LIN {X 0,Y 467.201,Z 533.915,A -85,B 0,C 180,E1 -7658.87,E2 -7658.87} C_VEL
LIN {X 0,Y 467.55,Z 525.583,A -85,B 0,C 180,E1 -7660.173,E2 -7660.173} C_VEL
LIN {X 0,Y 467.994,Z 517.028,A -85,B 0,C 180,E1 -7661.258,E2 -7661.258} C_VEL
LIN {X 0,Y 468.515,Z 506.992,A -85,B 0,C 180,E1 -7662.295,E2 -7662.295} C_VEL
LIN {X 0,Y 468.892,Z 496.03,A -85,B 0,C 180,E1 -7663.213,E2 -7663.213} C_VEL
LIN {X 0,Y 469.41,Z 484.584,A -85,B 0,C 180,E1 -7663.971,E2 -7663.971} C_VEL
LIN {X 0,Y 469.934,Z 471.495,A -85,B 0,C 180,E1 -7664.618,E2 -7664.618} C_VEL
LIN {X 0,Y 468.494,Z 459.642,A -85,B 0,C 180,E1 -7665.094,E2 -7665.094} C_VEL
LIN {X 0,Y 466.973,Z 449.848,A -85,B 0,C 180,E1 -7665.416,E2 -7665.416} C_VEL
LIN {X 0,Y 467.157,Z 441.535,A -85,B 0,C 180,E1 -7668.596,E2 -7668.596} C_VEL
LIN {X 0,Y 467.367,Z 433.791,A -85,B 0,C 180,E1 -7671.618,E2 -7671.618} C_VEL
LIN {X 0,Y 467.629,Z 425.59,A -85,B 0,C 180,E1 -7674.886,E2 -7674.886} C_VEL
LIN {X 0,Y 467.958,Z 417.432,A -85,B 0,C 180,E1 -7678.235,E2 -7678.235} C_VEL
LIN {X 0,Y 468.288,Z 410.455,A -85,B 0,C 180,E1 -7681.19,E2 -7681.19} C_VEL
LIN {X 0,Y 468.615,Z 404.693,A -85,B 0,C 180,E1 -7683.704,E2 -7683.704} C_VEL
LIN {X 0,Y 468.72,Z 399.752,A -85,B 0,C 180,E1 -7685.935,E2 -7685.935} C_VEL
LIN {X 0,Y 468.166,Z 395.47,A -85,B 0,C 180,E1 -7687.987,E2 -7687.987} C_VEL
LIN {X 0,Y 467.621,Z 392.239,A -85,B 0,C 180,E1 -7689.628,E2 -7689.628} C_VEL
LIN {X 0,Y 467.588,Z 392.243,A -85,B 0,C 180,E1 -7692.567,E2 -7692.567} C_VEL
LIN {X 0,Y 467.567,Z 392.245,A -85,B 0,C 180,E1 -7695.052,E2 -7695.052} C_VEL
LIN {X 0,Y 467.59,Z 392.242,A -85,B 0,C 180,E1 -7697.44,E2 -7697.44} C_VEL
LIN {X 0,Y 467.577,Z 392.245,A -85,B 0,C 180,E1 -7700.855,E2 -7700.855} C_VEL
LIN {X 0,Y 467.562,Z 392.244,A -85,B 0,C 180,E1 -7704.261,E2 -7704.261} C_VEL
LIN {X 0,Y 467.58,Z 392.243,A -85,B 0,C 180,E1 -7707.321,E2 -7707.321} C_VEL
LIN {X 0,Y 467.571,Z 392.244,A -85,B 0,C 180,E1 -7710.667,E2 -7710.667} C_VEL
LIN {X 0,Y 467.617,Z 392.238,A -85,B 0,C 180,E1 -7713.2,E2 -7713.2} C_VEL
LIN {X 0,Y 467.593,Z 392.241,A -85,B 0,C 180,E1 -7716.468,E2 -7716.468} C_VEL
LIN {X 0,Y 467.623,Z 392.237,A -85,B 0,C 180,E1 -7719.777,E2 -7719.777} C_VEL
LIN {X 0,Y 467.607,Z 392.24,A -85,B 0,C 180,E1 -7722.507,E2 -7722.507} C_VEL
LIN {X 0,Y 467.607,Z 392.24,A -85,B 0,C 180,E1 -7725.196,E2 -7725.196} C_VEL
LIN {X 0,Y 467.656,Z 392.233,A -85,B 0,C 180,E1 -7727.854,E2 -7727.854} C_VEL
LIN {X 0,Y 467.682,Z 392.231,A -85,B 0,C 180,E1 -7731.357,E2 -7731.357} C_VEL
LIN {X 0,Y 467.744,Z 392.221,A -85,B 0,C 180,E1 -7733.963,E2 -7733.963} C_VEL
LIN {X 0,Y 467.859,Z 392.209,A -85,B 0,C 180,E1 -7737.417,E2 -7737.417} C_VEL
LIN {X 0,Y 467.882,Z 392.204,A -85,B 0,C 180,E1 -7740,E2 -7740} C_VEL
LIN {X 0,Y 467.859,Z 392.21,A -85,B 0,C 180,E1 -7742.583,E2 -7742.583} C_VEL
LIN {X 0,Y 467.743,Z 392.222,A -85,B 0,C 180,E1 -7746.037,E2 -7746.037} C_VEL
LIN {X 0,Y 467.682,Z 392.231,A -85,B 0,C 180,E1 -7748.643,E2 -7748.643} C_VEL
LIN {X 0,Y 467.656,Z 392.233,A -85,B 0,C 180,E1 -7752.145,E2 -7752.145} C_VEL
LIN {X 0,Y 467.639,Z 392.234,A -85,B 0,C 180,E1 -7755.695,E2 -7755.695} C_VEL
LIN {X 0,Y 467.618,Z 392.239,A -85,B 0,C 180,E1 -7758.764,E2 -7758.764} C_VEL
LIN {X 0,Y 467.581,Z 392.244,A -85,B 0,C 180,E1 -7761.268,E2 -7761.268} C_VEL
LIN {X 0,Y 467.572,Z 392.243,A -85,B 0,C 180,E1 -7763.943,E2 -7763.943} C_VEL
LIN {X 0,Y 467.617,Z 392.238,A -85,B 0,C 180,E1 -7766.8,E2 -7766.8} C_VEL
LIN {X 0,Y 467.554,Z 392.245,A -85,B 0,C 180,E1 -7769.738,E2 -7769.738} C_VEL
LIN {X 0,Y 467.584,Z 392.243,A -85,B 0,C 180,E1 -7772.758,E2 -7772.758} C_VEL
LIN {X 0,Y 467.557,Z 392.245,A -85,B 0,C 180,E1 -7775.889,E2 -7775.889} C_VEL
LIN {X 0,Y 467.576,Z 392.244,A -85,B 0,C 180,E1 -7779.145,E2 -7779.145} C_VEL
LIN {X 0,Y 467.587,Z 392.242,A -85,B 0,C 180,E1 -7782.567,E2 -7782.567} C_VEL
LIN {X 0,Y 467.567,Z 392.245,A -85,B 0,C 180,E1 -7785.053,E2 -7785.053} C_VEL
LIN {X 0,Y 467.59,Z 392.241,A -85,B 0,C 180,E1 -7787.44,E2 -7787.44} C_VEL
LIN {X 0,Y 467.583,Z 392.243,A -85,B 0,C 180,E1 -7790.855,E2 -7790.855} C_VEL
LIN {X 0,Y 467.564,Z 392.245,A -85,B 0,C 180,E1 -7794.26,E2 -7794.26} C_VEL
LIN {X 0,Y 467.583,Z 392.242,A -85,B 0,C 180,E1 -7797.321,E2 -7797.321} C_VEL
LIN {X 0,Y 467.572,Z 392.245,A -85,B 0,C 180,E1 -7800.667,E2 -7800.667} C_VEL
LIN {X 0,Y 467.618,Z 392.238,A -85,B 0,C 180,E1 -7803.2,E2 -7803.2} C_VEL
LIN {X 0,Y 467.595,Z 392.241,A -85,B 0,C 180,E1 -7806.468,E2 -7806.468} C_VEL
LIN {X 0,Y 467.625,Z 392.236,A -85,B 0,C 180,E1 -7809.777,E2 -7809.777} C_VEL
LIN {X 0,Y 467.609,Z 392.24,A -85,B 0,C 180,E1 -7812.507,E2 -7812.507} C_VEL
LIN {X 0,Y 467.599,Z 392.239,A -85,B 0,C 180,E1 -7815.416,E2 -7815.416} C_VEL
LIN {X 0,Y 466.929,Z 392.325,A -85,B 0,C 180,E1 -7816.135,E2 -7816.135} C_VEL
LIN {X 0,Y 464.085,Z 392.677,A -85,B 0,C 180,E1 -7817.303,E2 -7817.303} C_VEL
LIN {X 0,Y 461.686,Z 392.977,A -85,B 0,C 180,E1 -7818.245,E2 -7818.245} C_VEL
LIN {X 0,Y 460.659,Z 393.104,A -85,B 0,C 180,E1 -7818.973,E2 -7818.973} C_VEL
LIN {X 0,Y 460.576,Z 393.112,A -85,B 0,C 180,E1 -7819.219,E2 -7819.219} C_VEL
LIN {X 0,Y 460.723,Z 393.098,A -85,B 0,C 180,E1 -7822.538,E2 -7822.538} C_VEL
LIN {X 0,Y 460.699,Z 393.1,A -85,B 0,C 180,E1 -7824.748,E2 -7824.748} C_VEL
LIN {X 0,Y 460.802,Z 393.086,A -85,B 0,C 180,E1 -7827.377,E2 -7827.377} C_VEL
LIN {X 0,Y 460.855,Z 393.081,A -85,B 0,C 180,E1 -7830,E2 -7830} C_VEL
LIN {X 0,Y 460.826,Z 393.084,A -85,B 0,C 180,E1 -7832.622,E2 -7832.622} C_VEL
LIN {X 0,Y 460.679,Z 393.103,A -85,B 0,C 180,E1 -7836.13,E2 -7836.13} C_VEL
LIN {X 0,Y 460.387,Z 393.141,A -85,B 0,C 180,E1 -7838.78,E2 -7838.78} C_VEL
LIN {X 0,Y 460.288,Z 393.863,A -85,B 0,C 180,E1 -7839.669,E2 -7839.669} C_VEL
LIN {X 0,Y 460.2,Z 397.277,A -85,B 0,C 180,E1 -7842.345,E2 -7842.345} C_VEL
LIN {X 0,Y 460.068,Z 401.733,A -85,B 0,C 180,E1 -7845.764,E2 -7845.764} C_VEL
LIN {X 0,Y 459.93,Z 405.642,A -85,B 0,C 180,E1 -7848.716,E2 -7848.716} C_VEL
LIN {X 0,Y 459.788,Z 409.438,A -85,B 0,C 180,E1 -7851.521,E2 -7851.521} C_VEL
LIN {X 0,Y 459.726,Z 413.312,A -85,B 0,C 180,E1 -7854.378,E2 -7854.378} C_VEL
LIN {X 0,Y 459.679,Z 417.601,A -85,B 0,C 180,E1 -7857.454,E2 -7857.454} C_VEL
LIN {X 0,Y 462.867,Z 432.273,A -85,B 0,C 180,E1 -7858.027,E2 -7858.027} C_VEL
LIN {X 0,Y 463.264,Z 437.27,A -85,B 0,C 180,E1 -7858.249,E2 -7858.249} C_VEL
LIN {X 0,Y 462.774,Z 449.809,A -85,B 0,C 180,E1 -7858.889,E2 -7858.889} C_VEL
LIN {X 0,Y 462.259,Z 460.524,A -85,B 0,C 180,E1 -7859.607,E2 -7859.607} C_VEL
LIN {X 0,Y 461.801,Z 471.37,A -85,B 0,C 180,E1 -7860.525,E2 -7860.525} C_VEL
LIN {X 0,Y 461.318,Z 481.28,A -85,B 0,C 180,E1 -7861.56,E2 -7861.56} C_VEL
LIN {X 0,Y 460.844,Z 490.462,A -85,B 0,C 180,E1 -7862.743,E2 -7862.743} C_VEL
LIN {X 0,Y 460.4,Z 499.041,A -85,B 0,C 180,E1 -7864.123,E2 -7864.123} C_VEL
LIN {X 0,Y 460.06,Z 505.812,A -85,B 0,C 180,E1 -7865.485,E2 -7865.485} C_VEL
LIN {X 0,Y 459.849,Z 511.567,A -85,B 0,C 180,E1 -7866.968,E2 -7866.968} C_VEL
LIN {X 0,Y 459.685,Z 515.328,A -85,B 0,C 180,E1 -7868.225,E2 -7868.225} C_VEL
LIN {X 0,Y 459.574,Z 517.956,A -85,B 0,C 180,E1 -7869.392,E2 -7869.392} C_VEL
LIN {X 0,Y 459.493,Z 519.215,A -85,B 0,C 180,E1 -7870.115,E2 -7870.115} C_VEL
LIN {X 0,Y 459.433,Z 520.788,A -85,B 0,C 180,E1 -7871.448,E2 -7871.448} C_VEL
LIN {X 0,Y 459.462,Z 521.432,A -85,B 0,C 180,E1 -7872.759,E2 -7872.759} C_VEL
LIN {X 0,Y 459.474,Z 521.217,A -85,B 0,C 180,E1 -7874.036,E2 -7874.036} C_VEL
LIN {X 0,Y 459.498,Z 520.204,A -85,B 0,C 180,E1 -7875.286,E2 -7875.286} C_VEL
LIN {X 0,Y 459.593,Z 518.401,A -85,B 0,C 180,E1 -7876.518,E2 -7876.518} C_VEL
LIN {X 0,Y 459.735,Z 514.685,A -85,B 0,C 180,E1 -7878.149,E2 -7878.149} C_VEL
LIN {X 0,Y 459.919,Z 509.247,A -85,B 0,C 180,E1 -7879.821,E2 -7879.821} C_VEL
LIN {X 0,Y 460.22,Z 503.109,A -85,B 0,C 180,E1 -7881.236,E2 -7881.236} C_VEL
LIN {X 0,Y 460.581,Z 496.18,A -85,B 0,C 180,E1 -7882.51,E2 -7882.51} C_VEL
LIN {X 0,Y 461.062,Z 486.859,A -85,B 0,C 180,E1 -7883.888,E2 -7883.888} C_VEL
LIN {X 0,Y 461.597,Z 477.131,A -85,B 0,C 180,E1 -7885.034,E2 -7885.034} C_VEL
LIN {X 0,Y 462.139,Z 466.904,A -85,B 0,C 180,E1 -7886.007,E2 -7886.007} C_VEL
LIN {X 0,Y 462.597,Z 456.021,A -85,B 0,C 180,E1 -7886.843,E2 -7886.843} C_VEL
LIN {X 0,Y 463.118,Z 444.532,A -85,B 0,C 180,E1 -7887.532,E2 -7887.532} C_VEL
LIN {X 0,Y 463.321,Z 434.551,A -85,B 0,C 180,E1 -7887.997,E2 -7887.997} C_VEL
LIN {X 0,Y 460.593,Z 421.943,A -85,B 0,C 180,E1 -7888.525,E2 -7888.525} C_VEL
LIN {X 0,Y 459.753,Z 418.131,A -85,B 0,C 180,E1 -7888.669,E2 -7888.669} C_VEL
LIN {X 0,Y 459.786,Z 414.027,A -85,B 0,C 180,E1 -7891.716,E2 -7891.716} C_VEL
LIN {X 0,Y 459.956,Z 410.111,A -85,B 0,C 180,E1 -7894.67,E2 -7894.67} C_VEL
LIN {X 0,Y 460.056,Z 406.354,A -85,B 0,C 180,E1 -7897.548,E2 -7897.548} C_VEL
LIN {X 0,Y 460.159,Z 402.747,A -85,B 0,C 180,E1 -7900.366,E2 -7900.366} C_VEL
LIN {X 0,Y 460.271,Z 399.284,A -85,B 0,C 180,E1 -7903.135,E2 -7903.135} C_VEL
LIN {X 0,Y 460.374,Z 395.891,A -85,B 0,C 180,E1 -7905.862,E2 -7905.862} C_VEL
LIN {X 0,Y 460.468,Z 393.714,A -85,B 0,C 180,E1 -7907.662,E2 -7907.662} C_VEL
LIN {X 0,Y 460.519,Z 393.124,A -85,B 0,C 180,E1 -7908.557,E2 -7908.557} C_VEL
LIN {X 0,Y 460.624,Z 393.114,A -85,B 0,C 180,E1 -7911.224,E2 -7911.224} C_VEL
LIN {X 0,Y 460.706,Z 393.099,A -85,B 0,C 180,E1 -7913.87,E2 -7913.87} C_VEL
LIN {X 0,Y 460.821,Z 393.086,A -85,B 0,C 180,E1 -7917.378,E2 -7917.378} C_VEL
LIN {X 0,Y 460.849,Z 393.082,A -85,B 0,C 180,E1 -7920,E2 -7920} C_VEL
LIN {X 0,Y 460.82,Z 393.084,A -85,B 0,C 180,E1 -7922.622,E2 -7922.622} C_VEL
LIN {X 0,Y 460.706,Z 393.1,A -85,B 0,C 180,E1 -7926.13,E2 -7926.13} C_VEL
LIN {X 0,Y 460.625,Z 393.11,A -85,B 0,C 180,E1 -7928.776,E2 -7928.776} C_VEL
LIN {X 0,Y 460.609,Z 393.112,A -85,B 0,C 180,E1 -7932.445,E2 -7932.445} C_VEL
LIN {X 0,Y 460.596,Z 393.113,A -85,B 0,C 180,E1 -7935.998,E2 -7935.998} C_VEL
LIN {X 0,Y 460.567,Z 393.116,A -85,B 0,C 180,E1 -7938.902,E2 -7938.902} C_VEL
LIN {X 0,Y 460.512,Z 393.124,A -85,B 0,C 180,E1 -7941.486,E2 -7941.486} C_VEL
LIN {X 0,Y 460.539,Z 393.118,A -85,B 0,C 180,E1 -7944.333,E2 -7944.333} C_VEL
LIN {X 0,Y 460.581,Z 393.115,A -85,B 0,C 180,E1 -7947.243,E2 -7947.243} C_VEL
LIN {X 0,Y 460.524,Z 393.122,A -85,B 0,C 180,E1 -7950.239,E2 -7950.239} C_VEL
LIN {X 0,Y 460.526,Z 393.122,A -85,B 0,C 180,E1 -7953.325,E2 -7953.325} C_VEL
LIN {X 0,Y 460.477,Z 393.129,A -85,B 0,C 180,E1 -7956.53,E2 -7956.53} C_VEL
LIN {X 0,Y 460.576,Z 393.117,A -85,B 0,C 180,E1 -7959.858,E2 -7959.858} C_VEL
LIN {X 0,Y 460.511,Z 393.125,A -85,B 0,C 180,E1 -7962.901,E2 -7962.901} C_VEL
LIN {X 0,Y 460.509,Z 393.124,A -85,B 0,C 180,E1 -7965.831,E2 -7965.831} C_VEL
LIN {X 0,Y 460.541,Z 393.119,A -85,B 0,C 180,E1 -7968.991,E2 -7968.991} C_VEL
LIN {X 0,Y 460.58,Z 393.173,A -85,B 0,C 180,E1 -7969.799,E2 -7969.799} C_VEL
LIN {X 0,Y 461.533,Z 399.106,A -85,B 0,C 180,E1 -7973.024,E2 -7973.024} C_VEL
LIN {X 0,Y 461.753,Z 403.631,A -85,B 0,C 180,E1 -7975.275,E2 -7975.275} C_VEL
LIN {X 0,Y 461.39,Z 408.979,A -85,B 0,C 180,E1 -7977.784,E2 -7977.784} C_VEL
LIN {X 0,Y 460.976,Z 415.748,A -85,B 0,C 180,E1 -7980.8,E2 -7980.8} C_VEL
LIN {X 0,Y 460.62,Z 423.684,A -85,B 0,C 180,E1 -7984.185,E2 -7984.185} C_VEL
LIN {X 0,Y 460.34,Z 431.917,A -85,B 0,C 180,E1 -7987.563,E2 -7987.563} C_VEL
LIN {X 0,Y 460.079,Z 440.121,A -85,B 0,C 180,E1 -7990.827,E2 -7990.827} C_VEL
LIN {X 0,Y 459.905,Z 448.373,A -85,B 0,C 180,E1 -7994.035,E2 -7994.035} C_VEL
LIN {X 0,Y 459.859,Z 449.138,A -85,B 0,C 180,E1 -7994.329,E2 -7994.329} C_VEL
LIN {X 0,Y 462.172,Z 464.362,A -85,B 0,C 180,E1 -7994.857,E2 -7994.857} C_VEL
LIN {X 0,Y 463.01,Z 472.453,A -85,B 0,C 180,E1 -7995.215,E2 -7995.215} C_VEL
LIN {X 0,Y 462.524,Z 484.144,A -85,B 0,C 180,E1 -7995.818,E2 -7995.818} C_VEL
LIN {X 0,Y 461.969,Z 495.547,A -85,B 0,C 180,E1 -7996.586,E2 -7996.586} C_VEL
LIN {X 0,Y 461.437,Z 506.673,A -85,B 0,C 180,E1 -7997.531,E2 -7997.531} C_VEL
LIN {X 0,Y 460.977,Z 516.553,A -85,B 0,C 180,E1 -7998.569,E2 -7998.569} C_VEL
LIN {X 0,Y 460.496,Z 525.123,A -85,B 0,C 180,E1 -7999.67,E2 -7999.67} C_VEL
LIN {X 0,Y 460.129,Z 533.481,A -85,B 0,C 180,E1 -8000.993,E2 -8000.993} C_VEL
LIN {X 0,Y 459.883,Z 540.226,A -85,B 0,C 180,E1 -8002.316,E2 -8002.316} C_VEL
LIN {X 0,Y 459.674,Z 546.407,A -85,B 0,C 180,E1 -8003.857,E2 -8003.857} C_VEL
LIN {X 0,Y 459.621,Z 550.425,A -85,B 0,C 180,E1 -8005.176,E2 -8005.176} C_VEL
LIN {X 0,Y 459.588,Z 553.396,A -85,B 0,C 180,E1 -8006.494,E2 -8006.494} C_VEL
LIN {X 0,Y 459.585,Z 554.812,A -85,B 0,C 180,E1 -8007.371,E2 -8007.371} C_VEL
LIN {X 0,Y 459.552,Z 556.446,A -85,B 0,C 180,E1 -8009.124,E2 -8009.124} C_VEL
LIN {X 0,Y 459.53,Z 556.67,A -85,B 0,C 180,E1 -8010,E2 -8010} C_VEL
LIN {X 0,Y 459.552,Z 556.459,A -85,B 0,C 180,E1 -8010.877,E2 -8010.877} C_VEL
LIN {X 0,Y 459.585,Z 554.857,A -85,B 0,C 180,E1 -8012.63,E2 -8012.63} C_VEL
LIN {X 0,Y 459.588,Z 553.453,A -85,B 0,C 180,E1 -8013.507,E2 -8013.507} C_VEL
LIN {X 0,Y 459.621,Z 550.502,A -85,B 0,C 180,E1 -8014.825,E2 -8014.825} C_VEL
LIN {X 0,Y 459.715,Z 545.46,A -85,B 0,C 180,E1 -8016.431,E2 -8016.431} C_VEL
LIN {X 0,Y 459.909,Z 539.328,A -85,B 0,C 180,E1 -8017.905,E2 -8017.905} C_VEL
LIN {X 0,Y 460.226,Z 532.379,A -85,B 0,C 180,E1 -8019.227,E2 -8019.227} C_VEL
LIN {X 0,Y 460.581,Z 523.669,A -85,B 0,C 180,E1 -8020.551,E2 -8020.551} C_VEL
LIN {X 0,Y 461.103,Z 514.757,A -85,B 0,C 180,E1 -8021.651,E2 -8021.651} C_VEL
LIN {X 0,Y 461.615,Z 504.111,A -85,B 0,C 180,E1 -8022.724,E2 -8022.724} C_VEL
LIN {X 0,Y 462.104,Z 492.682,A -85,B 0,C 180,E1 -8023.635,E2 -8023.635} C_VEL
LIN {X 0,Y 462.691,Z 480.292,A -85,B 0,C 180,E1 -8024.402,E2 -8024.402} C_VEL
LIN {X 0,Y 463.053,Z 471.128,A -85,B 0,C 180,E1 -8024.84,E2 -8024.84} C_VEL
LIN {X 0,Y 461.181,Z 457.798,A -85,B 0,C 180,E1 -8025.384,E2 -8025.384} C_VEL
LIN {X 0,Y 459.908,Z 449.618,A -85,B 0,C 180,E1 -8025.642,E2 -8025.642} C_VEL
LIN {X 0,Y 460.117,Z 440.704,A -85,B 0,C 180,E1 -8029.126,E2 -8029.126} C_VEL
LIN {X 0,Y 460.325,Z 433.575,A -85,B 0,C 180,E1 -8031.966,E2 -8031.966} C_VEL
LIN {X 0,Y 460.609,Z 425.402,A -85,B 0,C 180,E1 -8035.292,E2 -8035.292} C_VEL
LIN {X 0,Y 460.971,Z 417.26,A -85,B 0,C 180,E1 -8038.702,E2 -8038.702} C_VEL
LIN {X 0,Y 461.291,Z 410.929,A -85,B 0,C 180,E1 -8041.439,E2 -8041.439} C_VEL
LIN {X 0,Y 461.737,Z 403.563,A -85,B 0,C 180,E1 -8044.722,E2 -8044.722} C_VEL
LIN {X 0,Y 461.531,Z 398.786,A -85,B 0,C 180,E1 -8046.977,E2 -8046.977} C_VEL
LIN {X 0,Y 460.574,Z 393.117,A -85,B 0,C 180,E1 -8049.858,E2 -8049.858} C_VEL
LIN {X 0,Y 460.514,Z 393.123,A -85,B 0,C 180,E1 -8052.9,E2 -8052.9} C_VEL
LIN {X 0,Y 460.51,Z 393.125,A -85,B 0,C 180,E1 -8055.831,E2 -8055.831} C_VEL
LIN {X 0,Y 460.532,Z 393.121,A -85,B 0,C 180,E1 -8058.989,E2 -8058.989} C_VEL
LIN {X 0,Y 460.525,Z 393.122,A -85,B 0,C 180,E1 -8061.267,E2 -8061.267} C_VEL
LIN {X 0,Y 460.512,Z 393.123,A -85,B 0,C 180,E1 -8064.554,E2 -8064.554} C_VEL
LIN {X 0,Y 460.531,Z 393.121,A -85,B 0,C 180,E1 -8067.715,E2 -8067.715} C_VEL
LIN {X 0,Y 460.541,Z 393.12,A -85,B 0,C 180,E1 -8070.769,E2 -8070.769} C_VEL
LIN {X 0,Y 460.564,Z 393.116,A -85,B 0,C 180,E1 -8073.735,E2 -8073.735} C_VEL
LIN {X 0,Y 460.547,Z 393.119,A -85,B 0,C 180,E1 -8076.624,E2 -8076.624} C_VEL
LIN {X 0,Y 460.552,Z 393.119,A -85,B 0,C 180,E1 -8079.453,E2 -8079.453} C_VEL
LIN {X 0,Y 460.558,Z 393.117,A -85,B 0,C 180,E1 -8082.23,E2 -8082.23} C_VEL
LIN {X 0,Y 460.566,Z 393.117,A -85,B 0,C 180,E1 -8084.965,E2 -8084.965} C_VEL
LIN {X 0,Y 460.611,Z 393.111,A -85,B 0,C 180,E1 -8088.559,E2 -8088.559} C_VEL
LIN {X 0,Y 460.696,Z 393.099,A -85,B 0,C 180,E1 -8092.108,E2 -8092.108} C_VEL
LIN {X 0,Y 460.696,Z 393.1,A -85,B 0,C 180,E1 -8094.748,E2 -8094.748} C_VEL
LIN {X 0,Y 460.8,Z 393.088,A -85,B 0,C 180,E1 -8097.377,E2 -8097.377} C_VEL
LIN {X 0,Y 460.853,Z 393.08,A -85,B 0,C 180,E1 -8100,E2 -8100} C_VEL
LIN {X 0,Y 460.8,Z 393.089,A -85,B 0,C 180,E1 -8102.622,E2 -8102.622} C_VEL
LIN {X 0,Y 460.71,Z 393.098,A -85,B 0,C 180,E1 -8106.13,E2 -8106.13} C_VEL
LIN {X 0,Y 460.629,Z 393.109,A -85,B 0,C 180,E1 -8108.776,E2 -8108.776} C_VEL
LIN {X 0,Y 460.614,Z 393.111,A -85,B 0,C 180,E1 -8112.445,E2 -8112.445} C_VEL
LIN {X 0,Y 460.601,Z 393.111,A -85,B 0,C 180,E1 -8115.998,E2 -8115.998} C_VEL
LIN {X 0,Y 460.571,Z 393.117,A -85,B 0,C 180,E1 -8118.902,E2 -8118.902} C_VEL
LIN {X 0,Y 460.516,Z 393.122,A -85,B 0,C 180,E1 -8121.486,E2 -8121.486} C_VEL
LIN {X 0,Y 460.542,Z 393.12,A -85,B 0,C 180,E1 -8124.332,E2 -8124.332} C_VEL
LIN {X 0,Y 460.573,Z 393.116,A -85,B 0,C 180,E1 -8127.244,E2 -8127.244} C_VEL
LIN {X 0,Y 460.511,Z 393.124,A -85,B 0,C 180,E1 -8130.24,E2 -8130.24} C_VEL
LIN {X 0,Y 460.53,Z 393.121,A -85,B 0,C 180,E1 -8133.325,E2 -8133.325} C_VEL
LIN {X 0,Y 460.479,Z 393.127,A -85,B 0,C 180,E1 -8136.529,E2 -8136.529} C_VEL
LIN {X 0,Y 460.528,Z 393.12,A -85,B 0,C 180,E1 -8139.863,E2 -8139.863} C_VEL
LIN {X 0,Y 460.514,Z 393.124,A -85,B 0,C 180,E1 -8142.9,E2 -8142.9} C_VEL
LIN {X 0,Y 460.51,Z 393.123,A -85,B 0,C 180,E1 -8145.831,E2 -8145.831} C_VEL
LIN {X 0,Y 460.532,Z 393.121,A -85,B 0,C 180,E1 -8148.989,E2 -8148.989} C_VEL
LIN {X 0,Y 460.527,Z 393.121,A -85,B 0,C 180,E1 -8151.267,E2 -8151.267} C_VEL
LIN {X 0,Y 460.514,Z 393.124,A -85,B 0,C 180,E1 -8154.555,E2 -8154.555} C_VEL
LIN {X 0,Y 460.533,Z 393.12,A -85,B 0,C 180,E1 -8157.716,E2 -8157.716} C_VEL
LIN {X 0,Y 460.542,Z 393.121,A -85,B 0,C 180,E1 -8160.769,E2 -8160.769} C_VEL
LIN {X 0,Y 460.565,Z 393.116,A -85,B 0,C 180,E1 -8163.735,E2 -8163.735} C_VEL
LIN {X 0,Y 460.548,Z 393.12,A -85,B 0,C 180,E1 -8166.624,E2 -8166.624} C_VEL
LIN {X 0,Y 460.553,Z 393.117,A -85,B 0,C 180,E1 -8169.453,E2 -8169.453} C_VEL
LIN {X 0,Y 460.559,Z 393.117,A -85,B 0,C 180,E1 -8172.23,E2 -8172.23} C_VEL
LIN {X 0,Y 460.568,Z 393.117,A -85,B 0,C 180,E1 -8174.965,E2 -8174.965} C_VEL
LIN {X 0,Y 460.612,Z 393.112,A -85,B 0,C 180,E1 -8178.559,E2 -8178.559} C_VEL
LIN {X 0,Y 460.576,Z 393.112,A -85,B 0,C 180,E1 -8179.219,E2 -8179.219} C_VEL
LIN {X 0,Y 459.92,Z 393.197,A -85,B 0,C 180,E1 -8179.949,E2 -8179.949} C_VEL
LIN {X 0,Y 457.105,Z 393.547,A -85,B 0,C 180,E1 -8181.136,E2 -8181.136} C_VEL
LIN {X 0,Y 454.728,Z 393.844,A -85,B 0,C 180,E1 -8182.093,E2 -8182.093} C_VEL
LIN {X 0,Y 453.717,Z 393.969,A -85,B 0,C 180,E1 -8182.832,E2 -8182.832} C_VEL
LIN {X 0,Y 453.64,Z 393.977,A -85,B 0,C 180,E1 -8183.082,E2 -8183.082} C_VEL
LIN {X 0,Y 453.673,Z 393.976,A -85,B 0,C 180,E1 -8184.666,E2 -8184.666} C_VEL
LIN {X 0,Y 453.746,Z 393.965,A -85,B 0,C 180,E1 -8187.336,E2 -8187.336} C_VEL
LIN {X 0,Y 453.825,Z 393.956,A -85,B 0,C 180,E1 -8190,E2 -8190} C_VEL
LIN {X 0,Y 453.767,Z 393.964,A -85,B 0,C 180,E1 -8192.663,E2 -8192.663} C_VEL
LIN {X 0,Y 453.641,Z 393.979,A -85,B 0,C 180,E1 -8196.225,E2 -8196.225} C_VEL
LIN {X 0,Y 453.313,Z 394.022,A -85,B 0,C 180,E1 -8198.919,E2 -8198.919} C_VEL
LIN {X 0,Y 453.168,Z 396.002,A -85,B 0,C 180,E1 -8200.725,E2 -8200.725} C_VEL
LIN {X 0,Y 453.098,Z 399.471,A -85,B 0,C 180,E1 -8203.454,E2 -8203.454} C_VEL
LIN {X 0,Y 452.935,Z 403.058,A -85,B 0,C 180,E1 -8206.218,E2 -8206.218} C_VEL
LIN {X 0,Y 452.821,Z 406.756,A -85,B 0,C 180,E1 -8209.021,E2 -8209.021} C_VEL
LIN {X 0,Y 452.7,Z 410.561,A -85,B 0,C 180,E1 -8211.875,E2 -8211.875} C_VEL
LIN {X 0,Y 452.651,Z 414.507,A -85,B 0,C 180,E1 -8214.784,E2 -8214.784} C_VEL
LIN {X 0,Y 452.599,Z 417.813,A -85,B 0,C 180,E1 -8217.2,E2 -8217.2} C_VEL
LIN {X 0,Y 456.011,Z 433.552,A -85,B 0,C 180,E1 -8217.843,E2 -8217.843} C_VEL
LIN {X 0,Y 456.383,Z 437.928,A -85,B 0,C 180,E1 -8218.047,E2 -8218.047} C_VEL
LIN {X 0,Y 455.875,Z 449.998,A -85,B 0,C 180,E1 -8218.674,E2 -8218.674} C_VEL
LIN {X 0,Y 455.31,Z 461.602,A -85,B 0,C 180,E1 -8219.472,E2 -8219.472} C_VEL
LIN {X 0,Y 454.862,Z 471.75,A -85,B 0,C 180,E1 -8220.35,E2 -8220.35} C_VEL
LIN {X 0,Y 454.317,Z 481.996,A -85,B 0,C 180,E1 -8221.441,E2 -8221.441} C_VEL
LIN {X 0,Y 453.868,Z 490.484,A -85,B 0,C 180,E1 -8222.553,E2 -8222.553} C_VEL
LIN {X 0,Y 453.411,Z 498.904,A -85,B 0,C 180,E1 -8223.918,E2 -8223.918} C_VEL
LIN {X 0,Y 453.054,Z 505.74,A -85,B 0,C 180,E1 -8225.298,E2 -8225.298} C_VEL
LIN {X 0,Y 452.824,Z 511.214,A -85,B 0,C 180,E1 -8226.694,E2 -8226.694} C_VEL
LIN {X 0,Y 452.595,Z 516.179,A -85,B 0,C 180,E1 -8228.398,E2 -8228.398} C_VEL
LIN {X 0,Y 452.466,Z 518.637,A -85,B 0,C 180,E1 -8229.556,E2 -8229.556} C_VEL
LIN {X 0,Y 452.356,Z 520.366,A -85,B 0,C 180,E1 -8230.732,E2 -8230.732} C_VEL
LIN {X 0,Y 452.341,Z 521.396,A -85,B 0,C 180,E1 -8231.919,E2 -8231.919} C_VEL
LIN {X 0,Y 452.387,Z 521.748,A -85,B 0,C 180,E1 -8233.121,E2 -8233.121} C_VEL
LIN {X 0,Y 452.379,Z 521.317,A -85,B 0,C 180,E1 -8234.386,E2 -8234.386} C_VEL
LIN {X 0,Y 452.436,Z 520.069,A -85,B 0,C 180,E1 -8235.652,E2 -8235.652} C_VEL
LIN {X 0,Y 452.535,Z 518.052,A -85,B 0,C 180,E1 -8236.895,E2 -8236.895} C_VEL
LIN {X 0,Y 452.66,Z 515.102,A -85,B 0,C 180,E1 -8238.179,E2 -8238.179} C_VEL
LIN {X 0,Y 452.815,Z 511.032,A -85,B 0,C 180,E1 -8239.508,E2 -8239.508} C_VEL
LIN {X 0,Y 453.099,Z 505.737,A -85,B 0,C 180,E1 -8240.854,E2 -8240.854} C_VEL
LIN {X 0,Y 453.438,Z 498.942,A -85,B 0,C 180,E1 -8242.228,E2 -8242.228} C_VEL
LIN {X 0,Y 453.859,Z 491.28,A -85,B 0,C 180,E1 -8243.48,E2 -8243.48} C_VEL
LIN {X 0,Y 454.365,Z 482.232,A -85,B 0,C 180,E1 -8244.681,E2 -8244.681} C_VEL
LIN {X 0,Y 454.967,Z 471.593,A -85,B 0,C 180,E1 -8245.813,E2 -8245.813} C_VEL
LIN {X 0,Y 455.482,Z 461.711,A -85,B 0,C 180,E1 -8246.664,E2 -8246.664} C_VEL
LIN {X 0,Y 455.966,Z 450.849,A -85,B 0,C 180,E1 -8247.417,E2 -8247.417} C_VEL
LIN {X 0,Y 456.432,Z 439.403,A -85,B 0,C 180,E1 -8248.03,E2 -8248.03} C_VEL
LIN {X 0,Y 456.379,Z 434.991,A -85,B 0,C 180,E1 -8248.23,E2 -8248.23} C_VEL
LIN {X 0,Y 453.535,Z 422.238,A -85,B 0,C 180,E1 -8248.779,E2 -8248.779} C_VEL
LIN {X 0,Y 452.679,Z 418.434,A -85,B 0,C 180,E1 -8248.918,E2 -8248.918} C_VEL
LIN {X 0,Y 452.766,Z 414.026,A -85,B 0,C 180,E1 -8252.246,E2 -8252.246} C_VEL
LIN {X 0,Y 452.897,Z 410.115,A -85,B 0,C 180,E1 -8255.23,E2 -8255.23} C_VEL
LIN {X 0,Y 453.049,Z 405.876,A -85,B 0,C 180,E1 -8258.551,E2 -8258.551} C_VEL
LIN {X 0,Y 453.174,Z 401.64,A -85,B 0,C 180,E1 -8261.931,E2 -8261.931} C_VEL
LIN {X 0,Y 453.304,Z 398.22,A -85,B 0,C 180,E1 -8264.718,E2 -8264.718} C_VEL
LIN {X 0,Y 453.443,Z 394.834,A -85,B 0,C 180,E1 -8267.537,E2 -8267.537} C_VEL
LIN {X 0,Y 453.462,Z 394.004,A -85,B 0,C 180,E1 -8268.376,E2 -8268.376} C_VEL
LIN {X 0,Y 453.586,Z 393.99,A -85,B 0,C 180,E1 -8271.087,E2 -8271.087} C_VEL
LIN {X 0,Y 453.673,Z 393.976,A -85,B 0,C 180,E1 -8273.775,E2 -8273.775} C_VEL
LIN {X 0,Y 453.762,Z 393.966,A -85,B 0,C 180,E1 -8277.337,E2 -8277.337} C_VEL
LIN {X 0,Y 453.82,Z 393.957,A -85,B 0,C 180,E1 -8280,E2 -8280} C_VEL
LIN {X 0,Y 453.761,Z 393.964,A -85,B 0,C 180,E1 -8282.663,E2 -8282.663} C_VEL
LIN {X 0,Y 453.674,Z 393.976,A -85,B 0,C 180,E1 -8286.225,E2 -8286.225} C_VEL
LIN {X 0,Y 453.588,Z 393.987,A -85,B 0,C 180,E1 -8288.914,E2 -8288.914} C_VEL
LIN {X 0,Y 453.559,Z 393.99,A -85,B 0,C 180,E1 -8292.529,E2 -8292.529} C_VEL
LIN {X 0,Y 453.54,Z 393.992,A -85,B 0,C 180,E1 -8296.196,E2 -8296.196} C_VEL
LIN {X 0,Y 453.517,Z 393.995,A -85,B 0,C 180,E1 -8299.041,E2 -8299.041} C_VEL
LIN {X 0,Y 453.473,Z 394,A -85,B 0,C 180,E1 -8301.836,E2 -8301.836} C_VEL
LIN {X 0,Y 453.511,Z 393.996,A -85,B 0,C 180,E1 -8304.735,E2 -8304.735} C_VEL
LIN {X 0,Y 453.535,Z 393.993,A -85,B 0,C 180,E1 -8307.962,E2 -8307.962} C_VEL
LIN {X 0,Y 453.48,Z 394,A -85,B 0,C 180,E1 -8310.759,E2 -8310.759} C_VEL
LIN {X 0,Y 453.475,Z 394.002,A -85,B 0,C 180,E1 -8313.913,E2 -8313.913} C_VEL
LIN {X 0,Y 453.469,Z 394.004,A -85,B 0,C 180,E1 -8317.188,E2 -8317.188} C_VEL
LIN {X 0,Y 453.531,Z 393.996,A -85,B 0,C 180,E1 -8319.446,E2 -8319.446} C_VEL
LIN {X 0,Y 453.461,Z 394.003,A -85,B 0,C 180,E1 -8322.995,E2 -8322.995} C_VEL
LIN {X 0,Y 453.464,Z 394.001,A -85,B 0,C 180,E1 -8325.78,E2 -8325.78} C_VEL
LIN {X 0,Y 453.515,Z 393.996,A -85,B 0,C 180,E1 -8329.437,E2 -8329.437} C_VEL
LIN {X 0,Y 454.276,Z 398.627,A -85,B 0,C 180,E1 -8332.093,E2 -8332.093} C_VEL
LIN {X 0,Y 454.735,Z 402.336,A -85,B 0,C 180,E1 -8334.035,E2 -8334.035} C_VEL
LIN {X 0,Y 454.626,Z 406.706,A -85,B 0,C 180,E1 -8336.185,E2 -8336.185} C_VEL
LIN {X 0,Y 454.145,Z 413.391,A -85,B 0,C 180,E1 -8339.291,E2 -8339.291} C_VEL
LIN {X 0,Y 453.732,Z 420.174,A -85,B 0,C 180,E1 -8342.311,E2 -8342.311} C_VEL
LIN {X 0,Y 453.457,Z 427.086,A -85,B 0,C 180,E1 -8345.263,E2 -8345.263} C_VEL
LIN {X 0,Y 453.212,Z 434.909,A -85,B 0,C 180,E1 -8348.502,E2 -8348.502} C_VEL
LIN {X 0,Y 452.931,Z 443.402,A -85,B 0,C 180,E1 -8351.921,E2 -8351.921} C_VEL
LIN {X 0,Y 452.821,Z 448.958,A -85,B 0,C 180,E1 -8354.091,E2 -8354.091} C_VEL
LIN {X 0,Y 454.934,Z 462.32,A -85,B 0,C 180,E1 -8354.538,E2 -8354.538} C_VEL
LIN {X 0,Y 456.144,Z 472.291,A -85,B 0,C 180,E1 -8354.988,E2 -8354.988} C_VEL
LIN {X 0,Y 455.636,Z 483.938,A -85,B 0,C 180,E1 -8355.599,E2 -8355.599} C_VEL
LIN {X 0,Y 455.033,Z 495.319,A -85,B 0,C 180,E1 -8356.377,E2 -8356.377} C_VEL
LIN {X 0,Y 454.45,Z 506.649,A -85,B 0,C 180,E1 -8357.357,E2 -8357.357} C_VEL
LIN {X 0,Y 453.995,Z 516.291,A -85,B 0,C 180,E1 -8358.391,E2 -8358.391} C_VEL
LIN {X 0,Y 453.483,Z 524.848,A -85,B 0,C 180,E1 -8359.508,E2 -8359.508} C_VEL
LIN {X 0,Y 453.092,Z 533.2,A -85,B 0,C 180,E1 -8360.852,E2 -8360.852} C_VEL
LIN {X 0,Y 452.813,Z 539.943,A -85,B 0,C 180,E1 -8362.195,E2 -8362.195} C_VEL
LIN {X 0,Y 452.604,Z 546.128,A -85,B 0,C 180,E1 -8363.76,E2 -8363.76} C_VEL
LIN {X 0,Y 452.55,Z 550.149,A -85,B 0,C 180,E1 -8365.101,E2 -8365.101} C_VEL
LIN {X 0,Y 452.486,Z 553.121,A -85,B 0,C 180,E1 -8366.438,E2 -8366.438} C_VEL
LIN {X 0,Y 452.508,Z 554.539,A -85,B 0,C 180,E1 -8367.33,E2 -8367.33} C_VEL
LIN {X 0,Y 452.457,Z 556.175,A -85,B 0,C 180,E1 -8369.11,E2 -8369.11} C_VEL
LIN {X 0,Y 452.463,Z 556.4,A -85,B 0,C 180,E1 -8370,E2 -8370} C_VEL
LIN {X 0,Y 452.457,Z 556.186,A -85,B 0,C 180,E1 -8370.89,E2 -8370.89} C_VEL
LIN {X 0,Y 452.509,Z 554.584,A -85,B 0,C 180,E1 -8372.671,E2 -8372.671} C_VEL
LIN {X 0,Y 452.486,Z 553.177,A -85,B 0,C 180,E1 -8373.562,E2 -8373.562} C_VEL
LIN {X 0,Y 452.55,Z 550.224,A -85,B 0,C 180,E1 -8374.9,E2 -8374.9} C_VEL
LIN {X 0,Y 452.611,Z 545.67,A -85,B 0,C 180,E1 -8376.396,E2 -8376.396} C_VEL
LIN {X 0,Y 452.816,Z 540.054,A -85,B 0,C 180,E1 -8377.805,E2 -8377.805} C_VEL
LIN {X 0,Y 453.102,Z 533.325,A -85,B 0,C 180,E1 -8379.148,E2 -8379.148} C_VEL
LIN {X 0,Y 453.484,Z 524.978,A -85,B 0,C 180,E1 -8380.492,E2 -8380.492} C_VEL
LIN {X 0,Y 454.004,Z 516.402,A -85,B 0,C 180,E1 -8381.61,E2 -8381.61} C_VEL
LIN {X 0,Y 454.517,Z 506.795,A -85,B 0,C 180,E1 -8382.636,E2 -8382.636} C_VEL
LIN {X 0,Y 455.027,Z 495.369,A -85,B 0,C 180,E1 -8383.624,E2 -8383.624} C_VEL
LIN {X 0,Y 455.606,Z 483.888,A -85,B 0,C 180,E1 -8384.403,E2 -8384.403} C_VEL
LIN {X 0,Y 456.149,Z 472.038,A -85,B 0,C 180,E1 -8385.013,E2 -8385.013} C_VEL
LIN {X 0,Y 454.255,Z 458.402,A -85,B 0,C 180,E1 -8385.59,E2 -8385.59} C_VEL
LIN {X 0,Y 452.849,Z 449.412,A -85,B 0,C 180,E1 -8385.875,E2 -8385.875} C_VEL
LIN {X 0,Y 453.078,Z 440.364,A -85,B 0,C 180,E1 -8389.482,E2 -8389.482} C_VEL
LIN {X 0,Y 453.317,Z 432.201,A -85,B 0,C 180,E1 -8392.805,E2 -8392.805} C_VEL
LIN {X 0,Y 453.606,Z 424.473,A -85,B 0,C 180,E1 -8396.021,E2 -8396.021} C_VEL
LIN {X 0,Y 453.986,Z 417.08,A -85,B 0,C 180,E1 -8399.186,E2 -8399.186} C_VEL
LIN {X 0,Y 454.39,Z 410.153,A -85,B 0,C 180,E1 -8402.25,E2 -8402.25} C_VEL
LIN {X 0,Y 454.731,Z 404.132,A -85,B 0,C 180,E1 -8405.002,E2 -8405.002} C_VEL
LIN {X 0,Y 454.514,Z 399.783,A -85,B 0,C 180,E1 -8407.088,E2 -8407.088} C_VEL
LIN {X 0,Y 453.513,Z 393.996,A -85,B 0,C 180,E1 -8410.097,E2 -8410.097} C_VEL
LIN {X 0,Y 453.456,Z 394.003,A -85,B 0,C 180,E1 -8413.244,E2 -8413.244} C_VEL
LIN {X 0,Y 453.465,Z 394.003,A -85,B 0,C 180,E1 -8415.779,E2 -8415.779} C_VEL
LIN {X 0,Y 453.48,Z 393.998,A -85,B 0,C 180,E1 -8418.209,E2 -8418.209} C_VEL
LIN {X 0,Y 453.492,Z 393.998,A -85,B 0,C 180,E1 -8420.794,E2 -8420.794} C_VEL
LIN {X 0,Y 453.457,Z 394.001,A -85,B 0,C 180,E1 -8423.917,E2 -8423.917} C_VEL
LIN {X 0,Y 453.48,Z 393.999,A -85,B 0,C 180,E1 -8427.151,E2 -8427.151} C_VEL
LIN {X 0,Y 453.476,Z 393.999,A -85,B 0,C 180,E1 -8430.268,E2 -8430.268} C_VEL
LIN {X 0,Y 453.507,Z 393.996,A -85,B 0,C 180,E1 -8433.294,E2 -8433.294} C_VEL
LIN {X 0,Y 453.504,Z 393.995,A -85,B 0,C 180,E1 -8436.239,E2 -8436.239} C_VEL
LIN {X 0,Y 453.483,Z 393.999,A -85,B 0,C 180,E1 -8439.118,E2 -8439.118} C_VEL
LIN {X 0,Y 453.511,Z 393.994,A -85,B 0,C 180,E1 -8441.944,E2 -8441.944} C_VEL
LIN {X 0,Y 453.54,Z 393.993,A -85,B 0,C 180,E1 -8444.726,E2 -8444.726} C_VEL
LIN {X 0,Y 453.56,Z 393.989,A -85,B 0,C 180,E1 -8448.379,E2 -8448.379} C_VEL
LIN {X 0,Y 453.653,Z 393.976,A -85,B 0,C 180,E1 -8451.985,E2 -8451.985} C_VEL
LIN {X 0,Y 453.67,Z 393.975,A -85,B 0,C 180,E1 -8454.667,E2 -8454.667} C_VEL
LIN {X 0,Y 453.744,Z 393.967,A -85,B 0,C 180,E1 -8457.337,E2 -8457.337} C_VEL
LIN {X 0,Y 453.823,Z 393.955,A -85,B 0,C 180,E1 -8460,E2 -8460} C_VEL
LIN {X 0,Y 453.744,Z 393.968,A -85,B 0,C 180,E1 -8462.663,E2 -8462.663} C_VEL
LIN {X 0,Y 453.677,Z 393.974,A -85,B 0,C 180,E1 -8466.225,E2 -8466.225} C_VEL
LIN {X 0,Y 453.593,Z 393.985,A -85,B 0,C 180,E1 -8468.913,E2 -8468.913} C_VEL
LIN {X 0,Y 453.564,Z 393.989,A -85,B 0,C 180,E1 -8472.529,E2 -8472.529} C_VEL
LIN {X 0,Y 453.545,Z 393.99,A -85,B 0,C 180,E1 -8476.196,E2 -8476.196} C_VEL
LIN {X 0,Y 453.521,Z 393.996,A -85,B 0,C 180,E1 -8479.041,E2 -8479.041} C_VEL
LIN {X 0,Y 453.477,Z 393.998,A -85,B 0,C 180,E1 -8481.836,E2 -8481.836} C_VEL
LIN {X 0,Y 453.514,Z 393.995,A -85,B 0,C 180,E1 -8484.734,E2 -8484.734} C_VEL
LIN {X 0,Y 453.533,Z 393.991,A -85,B 0,C 180,E1 -8487.96,E2 -8487.96} C_VEL
LIN {X 0,Y 453.466,Z 393.998,A -85,B 0,C 180,E1 -8491.525,E2 -8491.525} C_VEL
LIN {X 0,Y 453.49,Z 393.999,A -85,B 0,C 180,E1 -8494.778,E2 -8494.778} C_VEL
LIN {X 0,Y 453.464,Z 394.002,A -85,B 0,C 180,E1 -8498.312,E2 -8498.312} C_VEL
LIN {X 0,Y 453.494,Z 393.999,A -85,B 0,C 180,E1 -8500.609,E2 -8500.609} C_VEL
LIN {X 0,Y 453.455,Z 394,A -85,B 0,C 180,E1 -8503.244,E2 -8503.244} C_VEL
LIN {X 0,Y 453.464,Z 394,A -85,B 0,C 180,E1 -8505.779,E2 -8505.779} C_VEL
LIN {X 0,Y 453.48,Z 393.999,A -85,B 0,C 180,E1 -8508.209,E2 -8508.209} C_VEL
LIN {X 0,Y 453.495,Z 393.997,A -85,B 0,C 180,E1 -8510.793,E2 -8510.793} C_VEL
LIN {X 0,Y 453.458,Z 394.002,A -85,B 0,C 180,E1 -8513.917,E2 -8513.917} C_VEL
LIN {X 0,Y 453.484,Z 393.998,A -85,B 0,C 180,E1 -8517.151,E2 -8517.151} C_VEL
LIN {X 0,Y 453.477,Z 394,A -85,B 0,C 180,E1 -8520.268,E2 -8520.268} C_VEL
LIN {X 0,Y 453.508,Z 393.994,A -85,B 0,C 180,E1 -8523.294,E2 -8523.294} C_VEL
LIN {X 0,Y 453.505,Z 393.996,A -85,B 0,C 180,E1 -8526.239,E2 -8526.239} C_VEL
LIN {X 0,Y 453.485,Z 393.998,A -85,B 0,C 180,E1 -8529.118,E2 -8529.118} C_VEL
LIN {X 0,Y 453.513,Z 393.996,A -85,B 0,C 180,E1 -8531.944,E2 -8531.944} C_VEL
LIN {X 0,Y 453.542,Z 393.992,A -85,B 0,C 180,E1 -8534.726,E2 -8534.726} C_VEL
LIN {X 0,Y 453.561,Z 393.99,A -85,B 0,C 180,E1 -8538.379,E2 -8538.379} C_VEL
LIN {X 0,Y 453.654,Z 393.977,A -85,B 0,C 180,E1 -8541.985,E2 -8541.985} C_VEL
LIN {X 0,Y 453.64,Z 393.977,A -85,B 0,C 180,E1 -8543.082,E2 -8543.082} C_VEL
LIN {X 0,Y 452.954,Z 394.065,A -85,B 0,C 180,E1 -8543.823,E2 -8543.823} C_VEL
LIN {X 0,Y 450.005,Z 394.43,A -85,B 0,C 180,E1 -8545.024,E2 -8545.024} C_VEL
LIN {X 0,Y 447.577,Z 394.735,A -85,B 0,C 180,E1 -8545.994,E2 -8545.994} C_VEL
LIN {X 0,Y 446.633,Z 394.853,A -85,B 0,C 180,E1 -8546.744,E2 -8546.744} C_VEL
LIN {X 0,Y 446.609,Z 394.853,A -85,B 0,C 180,E1 -8546.998,E2 -8546.998} C_VEL
LIN {X 0,Y 446.795,Z 394.832,A -85,B 0,C 180,E1 -8550,E2 -8550} C_VEL
LIN {X 0,Y 446.71,Z 394.843,A -85,B 0,C 180,E1 -8552.705,E2 -8552.705} C_VEL
LIN {X 0,Y 446.606,Z 394.856,A -85,B 0,C 180,E1 -8556.324,E2 -8556.324} C_VEL
LIN {X 0,Y 446.256,Z 394.9,A -85,B 0,C 180,E1 -8559.061,E2 -8559.061} C_VEL
LIN {X 0,Y 446.083,Z 398.869,A -85,B 0,C 180,E1 -8562.364,E2 -8562.364} C_VEL
LIN {X 0,Y 445.94,Z 402.918,A -85,B 0,C 180,E1 -8565.54,E2 -8565.54} C_VEL
LIN {X 0,Y 445.771,Z 407.313,A -85,B 0,C 180,E1 -8568.923,E2 -8568.923} C_VEL
LIN {X 0,Y 445.602,Z 411.704,A -85,B 0,C 180,E1 -8572.242,E2 -8572.242} C_VEL
LIN {X 0,Y 445.546,Z 415.671,A -85,B 0,C 180,E1 -8575.207,E2 -8575.207} C_VEL
LIN {X 0,Y 445.52,Z 418.085,A -85,B 0,C 180,E1 -8576.97,E2 -8576.97} C_VEL
LIN {X 0,Y 448.67,Z 432.627,A -85,B 0,C 180,E1 -8577.553,E2 -8577.553} C_VEL
LIN {X 0,Y 449.523,Z 437.234,A -85,B 0,C 180,E1 -8577.781,E2 -8577.781} C_VEL
LIN {X 0,Y 449.003,Z 449.455,A -85,B 0,C 180,E1 -8578.413,E2 -8578.413} C_VEL
LIN {X 0,Y 448.441,Z 460.914,A -85,B 0,C 180,E1 -8579.195,E2 -8579.195} C_VEL
LIN {X 0,Y 447.929,Z 471.75,A -85,B 0,C 180,E1 -8580.137,E2 -8580.137} C_VEL
LIN {X 0,Y 447.355,Z 481.888,A -85,B 0,C 180,E1 -8581.227,E2 -8581.227} C_VEL
LIN {X 0,Y 446.903,Z 490.211,A -85,B 0,C 180,E1 -8582.322,E2 -8582.322} C_VEL
LIN {X 0,Y 446.397,Z 498.753,A -85,B 0,C 180,E1 -8583.707,E2 -8583.707} C_VEL
LIN {X 0,Y 446.063,Z 505.117,A -85,B 0,C 180,E1 -8584.986,E2 -8584.986} C_VEL
LIN {X 0,Y 445.765,Z 511.041,A -85,B 0,C 180,E1 -8586.479,E2 -8586.479} C_VEL
LIN {X 0,Y 445.564,Z 515.545,A -85,B 0,C 180,E1 -8587.963,E2 -8587.963} C_VEL
LIN {X 0,Y 445.392,Z 518.634,A -85,B 0,C 180,E1 -8589.359,E2 -8589.359} C_VEL
LIN {X 0,Y 445.272,Z 520.69,A -85,B 0,C 180,E1 -8590.746,E2 -8590.746} C_VEL
LIN {X 0,Y 445.269,Z 521.777,A -85,B 0,C 180,E1 -8592.112,E2 -8592.112} C_VEL
LIN {X 0,Y 445.29,Z 521.813,A -85,B 0,C 180,E1 -8593.983,E2 -8593.983} C_VEL
LIN {X 0,Y 445.317,Z 520.892,A -85,B 0,C 180,E1 -8595.249,E2 -8595.249} C_VEL
LIN {X 0,Y 445.409,Z 519.114,A -85,B 0,C 180,E1 -8596.536,E2 -8596.536} C_VEL
LIN {X 0,Y 445.544,Z 516.43,A -85,B 0,C 180,E1 -8597.848,E2 -8597.848} C_VEL
LIN {X 0,Y 445.698,Z 512.713,A -85,B 0,C 180,E1 -8599.19,E2 -8599.19} C_VEL
LIN {X 0,Y 445.966,Z 507.832,A -85,B 0,C 180,E1 -8600.55,E2 -8600.55} C_VEL
LIN {X 0,Y 446.286,Z 501.547,A -85,B 0,C 180,E1 -8601.941,E2 -8601.941} C_VEL
LIN {X 0,Y 446.764,Z 493.531,A -85,B 0,C 180,E1 -8603.347,E2 -8603.347} C_VEL
LIN {X 0,Y 447.328,Z 484.262,A -85,B 0,C 180,E1 -8604.651,E2 -8604.651} C_VEL
LIN {X 0,Y 447.904,Z 474.419,A -85,B 0,C 180,E1 -8605.771,E2 -8605.771} C_VEL
LIN {X 0,Y 448.521,Z 463.745,A -85,B 0,C 180,E1 -8606.741,E2 -8606.741} C_VEL
LIN {X 0,Y 449.1,Z 451.758,A -85,B 0,C 180,E1 -8607.605,E2 -8607.605} C_VEL
LIN {X 0,Y 449.593,Z 440.135,A -85,B 0,C 180,E1 -8608.248,E2 -8608.248} C_VEL
LIN {X 0,Y 449.43,Z 435.623,A -85,B 0,C 180,E1 -8608.461,E2 -8608.461} C_VEL
LIN {X 0,Y 446.544,Z 422.662,A -85,B 0,C 180,E1 -8609.039,E2 -8609.039} C_VEL
LIN {X 0,Y 445.602,Z 418.722,A -85,B 0,C 180,E1 -8609.196,E2 -8609.196} C_VEL
LIN {X 0,Y 445.699,Z 414.02,A -85,B 0,C 180,E1 -8612.788,E2 -8612.788} C_VEL
LIN {X 0,Y 445.87,Z 409.774,A -85,B 0,C 180,E1 -8616.094,E2 -8616.094} C_VEL
LIN {X 0,Y 446.016,Z 406.419,A -85,B 0,C 180,E1 -8618.751,E2 -8618.751} C_VEL
LIN {X 0,Y 446.137,Z 402.865,A -85,B 0,C 180,E1 -8621.636,E2 -8621.636} C_VEL
LIN {X 0,Y 446.249,Z 399.451,A -85,B 0,C 180,E1 -8624.471,E2 -8624.471} C_VEL
LIN {X 0,Y 446.412,Z 395.916,A -85,B 0,C 180,E1 -8627.441,E2 -8627.441} C_VEL
LIN {X 0,Y 446.42,Z 395.053,A -85,B 0,C 180,E1 -8628.19,E2 -8628.19} C_VEL
LIN {X 0,Y 446.531,Z 394.869,A -85,B 0,C 180,E1 -8630.945,E2 -8630.945} C_VEL
LIN {X 0,Y 446.642,Z 394.852,A -85,B 0,C 180,E1 -8633.676,E2 -8633.676} C_VEL
LIN {X 0,Y 446.706,Z 394.844,A -85,B 0,C 180,E1 -8637.295,E2 -8637.295} C_VEL
LIN {X 0,Y 446.79,Z 394.833,A -85,B 0,C 180,E1 -8640,E2 -8640} C_VEL
LIN {X 0,Y 446.705,Z 394.843,A -85,B 0,C 180,E1 -8642.705,E2 -8642.705} C_VEL
LIN {X 0,Y 446.643,Z 394.851,A -85,B 0,C 180,E1 -8646.324,E2 -8646.324} C_VEL
LIN {X 0,Y 446.534,Z 394.866,A -85,B 0,C 180,E1 -8649.056,E2 -8649.056} C_VEL
LIN {X 0,Y 446.517,Z 394.867,A -85,B 0,C 180,E1 -8652.73,E2 -8652.73} C_VEL
LIN {X 0,Y 446.492,Z 394.87,A -85,B 0,C 180,E1 -8656.228,E2 -8656.228} C_VEL
LIN {X 0,Y 446.466,Z 394.874,A -85,B 0,C 180,E1 -8659.303,E2 -8659.303} C_VEL
LIN {X 0,Y 446.415,Z 394.879,A -85,B 0,C 180,E1 -8662.2,E2 -8662.2} C_VEL
LIN {X 0,Y 446.455,Z 394.874,A -85,B 0,C 180,E1 -8665.153,E2 -8665.153} C_VEL
LIN {X 0,Y 446.481,Z 394.871,A -85,B 0,C 180,E1 -8668.179,E2 -8668.179} C_VEL
LIN {X 0,Y 446.416,Z 394.879,A -85,B 0,C 180,E1 -8671.301,E2 -8671.301} C_VEL
LIN {X 0,Y 446.427,Z 394.878,A -85,B 0,C 180,E1 -8674.523,E2 -8674.523} C_VEL
LIN {X 0,Y 446.436,Z 394.88,A -85,B 0,C 180,E1 -8678.084,E2 -8678.084} C_VEL
LIN {X 0,Y 446.441,Z 394.878,A -85,B 0,C 180,E1 -8680.921,E2 -8680.921} C_VEL
LIN {X 0,Y 446.4,Z 394.882,A -85,B 0,C 180,E1 -8683.846,E2 -8683.846} C_VEL
LIN {X 0,Y 446.397,Z 394.883,A -85,B 0,C 180,E1 -8686.404,E2 -8686.404} C_VEL
LIN {X 0,Y 446.48,Z 395.05,A -85,B 0,C 180,E1 -8689.258,E2 -8689.258} C_VEL
LIN {X 0,Y 447.35,Z 400.18,A -85,B 0,C 180,E1 -8692.216,E2 -8692.216} C_VEL
LIN {X 0,Y 447.747,Z 404.476,A -85,B 0,C 180,E1 -8694.496,E2 -8694.496} C_VEL
LIN {X 0,Y 447.523,Z 408.84,A -85,B 0,C 180,E1 -8696.658,E2 -8696.658} C_VEL
LIN {X 0,Y 447.065,Z 415.615,A -85,B 0,C 180,E1 -8699.839,E2 -8699.839} C_VEL
LIN {X 0,Y 446.66,Z 422.312,A -85,B 0,C 180,E1 -8702.852,E2 -8702.852} C_VEL
LIN {X 0,Y 446.34,Z 429.513,A -85,B 0,C 180,E1 -8705.96,E2 -8705.96} C_VEL
LIN {X 0,Y 446.105,Z 436.16,A -85,B 0,C 180,E1 -8708.756,E2 -8708.756} C_VEL
LIN {X 0,Y 445.837,Z 444.339,A -85,B 0,C 180,E1 -8712.098,E2 -8712.098} C_VEL
LIN {X 0,Y 445.759,Z 448.56,A -85,B 0,C 180,E1 -8713.801,E2 -8713.801} C_VEL
LIN {X 0,Y 448.125,Z 463.837,A -85,B 0,C 180,E1 -8714.36,E2 -8714.36} C_VEL
LIN {X 0,Y 449.227,Z 473.343,A -85,B 0,C 180,E1 -8714.809,E2 -8714.809} C_VEL
LIN {X 0,Y 448.643,Z 485.491,A -85,B 0,C 180,E1 -8715.485,E2 -8715.485} C_VEL
LIN {X 0,Y 447.957,Z 497.942,A -85,B 0,C 180,E1 -8716.389,E2 -8716.389} C_VEL
LIN {X 0,Y 447.41,Z 508.906,A -85,B 0,C 180,E1 -8717.412,E2 -8717.412} C_VEL
LIN {X 0,Y 446.806,Z 519.653,A -85,B 0,C 180,E1 -8718.661,E2 -8718.661} C_VEL
LIN {X 0,Y 446.307,Z 527.594,A -85,B 0,C 180,E1 -8719.796,E2 -8719.796} C_VEL
LIN {X 0,Y 445.955,Z 535.366,A -85,B 0,C 180,E1 -8721.162,E2 -8721.162} C_VEL
LIN {X 0,Y 445.635,Z 542.532,A -85,B 0,C 180,E1 -8722.752,E2 -8722.752} C_VEL
LIN {X 0,Y 445.488,Z 546.73,A -85,B 0,C 180,E1 -8723.933,E2 -8723.933} C_VEL
LIN {X 0,Y 445.417,Z 550.963,A -85,B 0,C 180,E1 -8725.475,E2 -8725.475} C_VEL
LIN {X 0,Y 445.385,Z 552.85,A -85,B 0,C 180,E1 -8726.382,E2 -8726.382} C_VEL
LIN {X 0,Y 445.433,Z 554.269,A -85,B 0,C 180,E1 -8727.287,E2 -8727.287} C_VEL
LIN {X 0,Y 445.366,Z 555.904,A -85,B 0,C 180,E1 -8729.096,E2 -8729.096} C_VEL
LIN {X 0,Y 445.37,Z 556.128,A -85,B 0,C 180,E1 -8730,E2 -8730} C_VEL
LIN {X 0,Y 445.366,Z 555.914,A -85,B 0,C 180,E1 -8730.905,E2 -8730.905} C_VEL
LIN {X 0,Y 445.434,Z 554.311,A -85,B 0,C 180,E1 -8732.713,E2 -8732.713} C_VEL
LIN {X 0,Y 445.385,Z 552.9,A -85,B 0,C 180,E1 -8733.619,E2 -8733.619} C_VEL
LIN {X 0,Y 445.479,Z 549.945,A -85,B 0,C 180,E1 -8734.978,E2 -8734.978} C_VEL
LIN {X 0,Y 445.56,Z 544.485,A -85,B 0,C 180,E1 -8736.749,E2 -8736.749} C_VEL
LIN {X 0,Y 445.793,Z 538.742,A -85,B 0,C 180,E1 -8738.157,E2 -8738.157} C_VEL
LIN {X 0,Y 446.139,Z 531.774,A -85,B 0,C 180,E1 -8739.521,E2 -8739.521} C_VEL
LIN {X 0,Y 446.555,Z 523.035,A -85,B 0,C 180,E1 -8740.886,E2 -8740.886} C_VEL
LIN {X 0,Y 447.151,Z 514.098,A -85,B 0,C 180,E1 -8742.02,E2 -8742.02} C_VEL
LIN {X 0,Y 447.612,Z 504.057,A -85,B 0,C 180,E1 -8743.066,E2 -8743.066} C_VEL
LIN {X 0,Y 448.19,Z 493.509,A -85,B 0,C 180,E1 -8743.951,E2 -8743.951} C_VEL
LIN {X 0,Y 448.816,Z 481.46,A -85,B 0,C 180,E1 -8744.742,E2 -8744.742} C_VEL
LIN {X 0,Y 449.062,Z 471.514,A -85,B 0,C 180,E1 -8745.256,E2 -8745.256} C_VEL
LIN {X 0,Y 447.186,Z 457.939,A -85,B 0,C 180,E1 -8745.838,E2 -8745.838} C_VEL
LIN {X 0,Y 445.776,Z 449.141,A -85,B 0,C 180,E1 -8746.136,E2 -8746.136} C_VEL
LIN {X 0,Y 446.029,Z 440.115,A -85,B 0,C 180,E1 -8749.802,E2 -8749.802} C_VEL
LIN {X 0,Y 446.256,Z 433.143,A -85,B 0,C 180,E1 -8752.696,E2 -8752.696} C_VEL
LIN {X 0,Y 446.53,Z 426.156,A -85,B 0,C 180,E1 -8755.647,E2 -8755.647} C_VEL
LIN {X 0,Y 446.907,Z 419.206,A -85,B 0,C 180,E1 -8758.67,E2 -8758.67} C_VEL
LIN {X 0,Y 447.321,Z 411.844,A -85,B 0,C 180,E1 -8761.96,E2 -8761.96} C_VEL
LIN {X 0,Y 447.657,Z 406.527,A -85,B 0,C 180,E1 -8764.415,E2 -8764.415} C_VEL
LIN {X 0,Y 447.699,Z 403.07,A -85,B 0,C 180,E1 -8766.063,E2 -8766.063} C_VEL
LIN {X 0,Y 446.92,Z 397.329,A -85,B 0,C 180,E1 -8768.978,E2 -8768.978} C_VEL
LIN {X 0,Y 446.479,Z 394.872,A -85,B 0,C 180,E1 -8770.33,E2 -8770.33} C_VEL
LIN {X 0,Y 446.4,Z 394.883,A -85,B 0,C 180,E1 -8773.596,E2 -8773.596} C_VEL
LIN {X 0,Y 446.399,Z 394.88,A -85,B 0,C 180,E1 -8776.403,E2 -8776.403} C_VEL
LIN {X 0,Y 446.428,Z 394.878,A -85,B 0,C 180,E1 -8779.082,E2 -8779.082} C_VEL
LIN {X 0,Y 446.41,Z 394.878,A -85,B 0,C 180,E1 -8782.121,E2 -8782.121} C_VEL
LIN {X 0,Y 446.429,Z 394.878,A -85,B 0,C 180,E1 -8785.477,E2 -8785.477} C_VEL
LIN {X 0,Y 446.416,Z 394.878,A -85,B 0,C 180,E1 -8788.7,E2 -8788.7} C_VEL
LIN {X 0,Y 446.486,Z 394.868,A -85,B 0,C 180,E1 -8791.821,E2 -8791.821} C_VEL
LIN {X 0,Y 446.458,Z 394.874,A -85,B 0,C 180,E1 -8794.848,E2 -8794.848} C_VEL
LIN {X 0,Y 446.449,Z 394.873,A -85,B 0,C 180,E1 -8798.245,E2 -8798.245} C_VEL
LIN {X 0,Y 446.457,Z 394.874,A -85,B 0,C 180,E1 -8801.649,E2 -8801.649} C_VEL
LIN {X 0,Y 446.508,Z 394.867,A -85,B 0,C 180,E1 -8804.48,E2 -8804.48} C_VEL
LIN {X 0,Y 446.518,Z 394.865,A -85,B 0,C 180,E1 -8808.193,E2 -8808.193} C_VEL
LIN {X 0,Y 446.601,Z 394.854,A -85,B 0,C 180,E1 -8811.858,E2 -8811.858} C_VEL
LIN {X 0,Y 446.645,Z 394.851,A -85,B 0,C 180,E1 -8814.583,E2 -8814.583} C_VEL
LIN {X 0,Y 446.664,Z 394.847,A -85,B 0,C 180,E1 -8818.197,E2 -8818.197} C_VEL
LIN {X 0,Y 446.793,Z 394.831,A -85,B 0,C 180,E1 -8820,E2 -8820} C_VEL
LIN {X 0,Y 446.691,Z 394.846,A -85,B 0,C 180,E1 -8822.705,E2 -8822.705} C_VEL
LIN {X 0,Y 446.647,Z 394.85,A -85,B 0,C 180,E1 -8826.324,E2 -8826.324} C_VEL
LIN {X 0,Y 446.538,Z 394.864,A -85,B 0,C 180,E1 -8829.055,E2 -8829.055} C_VEL
LIN {X 0,Y 446.522,Z 394.866,A -85,B 0,C 180,E1 -8832.73,E2 -8832.73} C_VEL
LIN {X 0,Y 446.497,Z 394.868,A -85,B 0,C 180,E1 -8836.228,E2 -8836.228} C_VEL
LIN {X 0,Y 446.47,Z 394.871,A -85,B 0,C 180,E1 -8839.303,E2 -8839.303} C_VEL
LIN {X 0,Y 446.418,Z 394.878,A -85,B 0,C 180,E1 -8842.2,E2 -8842.2} C_VEL
LIN {X 0,Y 446.458,Z 394.874,A -85,B 0,C 180,E1 -8845.152,E2 -8845.152} C_VEL
LIN {X 0,Y 446.485,Z 394.869,A -85,B 0,C 180,E1 -8848.179,E2 -8848.179} C_VEL
LIN {X 0,Y 446.42,Z 394.876,A -85,B 0,C 180,E1 -8851.775,E2 -8851.775} C_VEL
LIN {X 0,Y 446.431,Z 394.878,A -85,B 0,C 180,E1 -8854.523,E2 -8854.523} C_VEL
LIN {X 0,Y 446.416,Z 394.878,A -85,B 0,C 180,E1 -8858.079,E2 -8858.079} C_VEL
LIN {X 0,Y 446.427,Z 394.878,A -85,B 0,C 180,E1 -8860.918,E2 -8860.918} C_VEL
LIN {X 0,Y 446.401,Z 394.878,A -85,B 0,C 180,E1 -8863.846,E2 -8863.846} C_VEL
LIN {X 0,Y 446.399,Z 394.882,A -85,B 0,C 180,E1 -8866.403,E2 -8866.403} C_VEL
LIN {X 0,Y 446.428,Z 394.876,A -85,B 0,C 180,E1 -8869.082,E2 -8869.082} C_VEL
LIN {X 0,Y 446.429,Z 394.877,A -85,B 0,C 180,E1 -8872.123,E2 -8872.123} C_VEL
LIN {X 0,Y 446.432,Z 394.874,A -85,B 0,C 180,E1 -8875.477,E2 -8875.477} C_VEL
LIN {X 0,Y 446.418,Z 394.879,A -85,B 0,C 180,E1 -8878.7,E2 -8878.7} C_VEL
LIN {X 0,Y 446.486,Z 394.868,A -85,B 0,C 180,E1 -8881.821,E2 -8881.821} C_VEL
LIN {X 0,Y 446.46,Z 394.873,A -85,B 0,C 180,E1 -8884.848,E2 -8884.848} C_VEL
LIN {X 0,Y 446.45,Z 394.876,A -85,B 0,C 180,E1 -8888.245,E2 -8888.245} C_VEL
LIN {X 0,Y 446.459,Z 394.873,A -85,B 0,C 180,E1 -8891.649,E2 -8891.649} C_VEL
LIN {X 0,Y 446.51,Z 394.868,A -85,B 0,C 180,E1 -8894.48,E2 -8894.48} C_VEL
LIN {X 0,Y 446.519,Z 394.866,A -85,B 0,C 180,E1 -8898.193,E2 -8898.193} C_VEL
LIN {X 0,Y 446.602,Z 394.855,A -85,B 0,C 180,E1 -8901.858,E2 -8901.858} C_VEL
LIN {X 0,Y 446.648,Z 394.852,A -85,B 0,C 180,E1 -8904.582,E2 -8904.582} C_VEL
LIN {X 0,Y 446.609,Z 394.853,A -85,B 0,C 180,E1 -8906.998,E2 -8906.998} C_VEL
LIN {X 0,Y 446.083,Z 394.92,A -85,B 0,C 180,E1 -8907.751,E2 -8907.751} C_VEL
LIN {X 0,Y 443.263,Z 395.273,A -85,B 0,C 180,E1 -8908.974,E2 -8908.974} C_VEL
LIN {X 0,Y 440.783,Z 395.582,A -85,B 0,C 180,E1 -8909.961,E2 -8909.961} C_VEL
LIN {X 0,Y 439.702,Z 395.715,A -85,B 0,C 180,E1 -8910.724,E2 -8910.724} C_VEL
LIN {X 0,Y 439.611,Z 395.724,A -85,B 0,C 180,E1 -8910.983,E2 -8910.983} C_VEL
LIN {X 0,Y 439.657,Z 395.721,A -85,B 0,C 180,E1 -8912.748,E2 -8912.748} C_VEL
LIN {X 0,Y 439.608,Z 395.726,A -85,B 0,C 180,E1 -8915.504,E2 -8915.504} C_VEL
LIN {X 0,Y 439.316,Z 395.765,A -85,B 0,C 180,E1 -8918.278,E2 -8918.278} C_VEL
LIN {X 0,Y 439.176,Z 395.782,A -85,B 0,C 180,E1 -8919.208,E2 -8919.208} C_VEL
LIN {X 0,Y 439.025,Z 399.747,A -85,B 0,C 180,E1 -8922.446,E2 -8922.446} C_VEL
LIN {X 0,Y 438.856,Z 404.344,A -85,B 0,C 180,E1 -8926.083,E2 -8926.083} C_VEL
LIN {X 0,Y 438.647,Z 408.978,A -85,B 0,C 180,E1 -8929.661,E2 -8929.661} C_VEL
LIN {X 0,Y 438.549,Z 412.852,A -85,B 0,C 180,E1 -8932.619,E2 -8932.619} C_VEL
LIN {X 0,Y 438.451,Z 416.892,A -85,B 0,C 180,E1 -8935.644,E2 -8935.644} C_VEL
LIN {X 0,Y 438.441,Z 418.31,A -85,B 0,C 180,E1 -8936.7,E2 -8936.7} C_VEL
LIN {X 0,Y 441.795,Z 433.558,A -85,B 0,C 180,E1 -8937.344,E2 -8937.344} C_VEL
LIN {X 0,Y 442.66,Z 438.718,A -85,B 0,C 180,E1 -8937.606,E2 -8937.606} C_VEL
LIN {X 0,Y 442.059,Z 451.311,A -85,B 0,C 180,E1 -8938.292,E2 -8938.292} C_VEL
LIN {X 0,Y 441.461,Z 462.644,A -85,B 0,C 180,E1 -8939.106,E2 -8939.106} C_VEL
LIN {X 0,Y 440.911,Z 473.989,A -85,B 0,C 180,E1 -8940.138,E2 -8940.138} C_VEL
LIN {X 0,Y 440.331,Z 483.731,A -85,B 0,C 180,E1 -8941.246,E2 -8941.246} C_VEL
LIN {X 0,Y 439.783,Z 492.634,A -85,B 0,C 180,E1 -8942.492,E2 -8942.492} C_VEL
LIN {X 0,Y 439.34,Z 499.783,A -85,B 0,C 180,E1 -8943.713,E2 -8943.713} C_VEL
LIN {X 0,Y 438.927,Z 507.064,A -85,B 0,C 180,E1 -8945.254,E2 -8945.254} C_VEL
LIN {X 0,Y 438.636,Z 512.561,A -85,B 0,C 180,E1 -8946.763,E2 -8946.763} C_VEL
LIN {X 0,Y 438.431,Z 516.643,A -85,B 0,C 180,E1 -8948.236,E2 -8948.236} C_VEL
LIN {X 0,Y 438.236,Z 519.875,A -85,B 0,C 180,E1 -8949.901,E2 -8949.901} C_VEL
LIN {X 0,Y 438.175,Z 521.357,A -85,B 0,C 180,E1 -8951.117,E2 -8951.117} C_VEL
LIN {X 0,Y 438.202,Z 522.19,A -85,B 0,C 180,E1 -8952.459,E2 -8952.459} C_VEL
LIN {X 0,Y 438.201,Z 522.182,A -85,B 0,C 180,E1 -8953.803,E2 -8953.803} C_VEL
LIN {X 0,Y 438.223,Z 521.325,A -85,B 0,C 180,E1 -8955.118,E2 -8955.118} C_VEL
LIN {X 0,Y 438.317,Z 519.682,A -85,B 0,C 180,E1 -8956.412,E2 -8956.412} C_VEL
LIN {X 0,Y 438.471,Z 517.268,A -85,B 0,C 180,E1 -8957.686,E2 -8957.686} C_VEL
LIN {X 0,Y 438.592,Z 514.11,A -85,B 0,C 180,E1 -8958.93,E2 -8958.93} C_VEL
LIN {X 0,Y 438.906,Z 508.682,A -85,B 0,C 180,E1 -8960.53,E2 -8960.53} C_VEL
LIN {X 0,Y 439.28,Z 501.749,A -85,B 0,C 180,E1 -8962.106,E2 -8962.106} C_VEL
LIN {X 0,Y 439.73,Z 494.474,A -85,B 0,C 180,E1 -8963.415,E2 -8963.415} C_VEL
LIN {X 0,Y 440.333,Z 485.453,A -85,B 0,C 180,E1 -8964.723,E2 -8964.723} C_VEL
LIN {X 0,Y 440.902,Z 476.628,A -85,B 0,C 180,E1 -8965.772,E2 -8965.772} C_VEL
LIN {X 0,Y 441.571,Z 465.675,A -85,B 0,C 180,E1 -8966.831,E2 -8966.831} C_VEL
LIN {X 0,Y 442.087,Z 454.482,A -85,B 0,C 180,E1 -8967.687,E2 -8967.687} C_VEL
LIN {X 0,Y 442.735,Z 442.148,A -85,B 0,C 180,E1 -8968.41,E2 -8968.41} C_VEL
LIN {X 0,Y 442.623,Z 436.962,A -85,B 0,C 180,E1 -8968.667,E2 -8968.667} C_VEL
LIN {X 0,Y 439.78,Z 424.182,A -85,B 0,C 180,E1 -8969.271,E2 -8969.271} C_VEL
LIN {X 0,Y 438.534,Z 419.028,A -85,B 0,C 180,E1 -8969.469,E2 -8969.469} C_VEL
LIN {X 0,Y 438.629,Z 415.349,A -85,B 0,C 180,E1 -8972.312,E2 -8972.312} C_VEL
LIN {X 0,Y 438.823,Z 410.787,A -85,B 0,C 180,E1 -8975.906,E2 -8975.906} C_VEL
LIN {X 0,Y 438.964,Z 406.504,A -85,B 0,C 180,E1 -8979.376,E2 -8979.376} C_VEL
LIN {X 0,Y 439.108,Z 402.94,A -85,B 0,C 180,E1 -8982.296,E2 -8982.296} C_VEL
LIN {X 0,Y 439.23,Z 399.546,A -85,B 0,C 180,E1 -8985.166,E2 -8985.166} C_VEL
LIN {X 0,Y 439.39,Z 396.269,A -85,B 0,C 180,E1 -8987.999,E2 -8987.999} C_VEL
LIN {X 0,Y 439.369,Z 395.759,A -85,B 0,C 180,E1 -8988.934,E2 -8988.934} C_VEL
LIN {X 0,Y 439.616,Z 395.729,A -85,B 0,C 180,E1 -8992.376,E2 -8992.376} C_VEL
LIN {X 0,Y 439.617,Z 395.728,A -85,B 0,C 180,E1 -8994.496,E2 -8994.496} C_VEL
LIN {X 0,Y 439.632,Z 395.726,A -85,B 0,C 180,E1 -8998.168,E2 -8998.168} C_VEL
LIN {X 0,Y 439.761,Z 395.709,A -85,B 0,C 180,E1 -9000,E2 -9000} C_VEL
LIN {X 0,Y 439.652,Z 395.722,A -85,B 0,C 180,E1 -9002.749,E2 -9002.749} C_VEL
LIN {X 0,Y 439.614,Z 395.727,A -85,B 0,C 180,E1 -9006.425,E2 -9006.425} C_VEL
LIN {X 0,Y 439.496,Z 395.742,A -85,B 0,C 180,E1 -9009.202,E2 -9009.202} C_VEL
LIN {X 0,Y 439.461,Z 395.746,A -85,B 0,C 180,E1 -9012.938,E2 -9012.938} C_VEL
LIN {X 0,Y 439.443,Z 395.749,A -85,B 0,C 180,E1 -9016.349,E2 -9016.349} C_VEL
LIN {X 0,Y 439.399,Z 395.753,A -85,B 0,C 180,E1 -9019.627,E2 -9019.627} C_VEL
LIN {X 0,Y 439.361,Z 395.759,A -85,B 0,C 180,E1 -9022.576,E2 -9022.576} C_VEL
LIN {X 0,Y 439.402,Z 395.754,A -85,B 0,C 180,E1 -9025.585,E2 -9025.585} C_VEL
LIN {X 0,Y 439.422,Z 395.751,A -85,B 0,C 180,E1 -9028.673,E2 -9028.673} C_VEL
LIN {X 0,Y 439.371,Z 395.758,A -85,B 0,C 180,E1 -9031.861,E2 -9031.861} C_VEL
LIN {X 0,Y 439.398,Z 395.756,A -85,B 0,C 180,E1 -9035.156,E2 -9035.156} C_VEL
LIN {X 0,Y 439.397,Z 395.756,A -85,B 0,C 180,E1 -9038.594,E2 -9038.594} C_VEL
LIN {X 0,Y 439.396,Z 395.757,A -85,B 0,C 180,E1 -9041.259,E2 -9041.259} C_VEL
LIN {X 0,Y 439.399,Z 395.754,A -85,B 0,C 180,E1 -9044.73,E2 -9044.73} C_VEL
LIN {X 0,Y 439.396,Z 395.752,A -85,B 0,C 180,E1 -9047.796,E2 -9047.796} C_VEL
LIN {X 0,Y 439.416,Z 395.906,A -85,B 0,C 180,E1 -9048.922,E2 -9048.922} C_VEL
LIN {X 0,Y 440.353,Z 401.263,A -85,B 0,C 180,E1 -9052.088,E2 -9052.088} C_VEL
LIN {X 0,Y 440.743,Z 405.529,A -85,B 0,C 180,E1 -9054.414,E2 -9054.414} C_VEL
LIN {X 0,Y 440.535,Z 409.872,A -85,B 0,C 180,E1 -9056.607,E2 -9056.607} C_VEL
LIN {X 0,Y 440.056,Z 416.102,A -85,B 0,C 180,E1 -9059.589,E2 -9059.589} C_VEL
LIN {X 0,Y 439.654,Z 422.18,A -85,B 0,C 180,E1 -9062.383,E2 -9062.383} C_VEL
LIN {X 0,Y 439.312,Z 429.816,A -85,B 0,C 180,E1 -9065.766,E2 -9065.766} C_VEL
LIN {X 0,Y 439.039,Z 437.11,A -85,B 0,C 180,E1 -9068.89,E2 -9068.89} C_VEL
LIN {X 0,Y 438.745,Z 445.267,A -85,B 0,C 180,E1 -9072.281,E2 -9072.281} C_VEL
LIN {X 0,Y 438.72,Z 448.322,A -85,B 0,C 180,E1 -9073.539,E2 -9073.539} C_VEL
LIN {X 0,Y 440.87,Z 461.794,A -85,B 0,C 180,E1 -9074.015,E2 -9074.015} C_VEL
LIN {X 0,Y 442.314,Z 474.332,A -85,B 0,C 180,E1 -9074.625,E2 -9074.625} C_VEL
LIN {X 0,Y 441.682,Z 487.058,A -85,B 0,C 180,E1 -9075.369,E2 -9075.369} C_VEL
LIN {X 0,Y 440.963,Z 498.813,A -85,B 0,C 180,E1 -9076.266,E2 -9076.266} C_VEL
LIN {X 0,Y 440.393,Z 509.738,A -85,B 0,C 180,E1 -9077.325,E2 -9077.325} C_VEL
LIN {X 0,Y 439.822,Z 519.404,A -85,B 0,C 180,E1 -9078.479,E2 -9078.479} C_VEL
LIN {X 0,Y 439.287,Z 527.341,A -85,B 0,C 180,E1 -9079.632,E2 -9079.632} C_VEL
LIN {X 0,Y 438.883,Z 535.106,A -85,B 0,C 180,E1 -9081.018,E2 -9081.018} C_VEL
LIN {X 0,Y 438.554,Z 542.273,A -85,B 0,C 180,E1 -9082.635,E2 -9082.635} C_VEL
LIN {X 0,Y 438.387,Z 546.907,A -85,B 0,C 180,E1 -9083.975,E2 -9083.975} C_VEL
LIN {X 0,Y 438.346,Z 550.701,A -85,B 0,C 180,E1 -9085.402,E2 -9085.402} C_VEL
LIN {X 0,Y 438.286,Z 552.585,A -85,B 0,C 180,E1 -9086.323,E2 -9086.323} C_VEL
LIN {X 0,Y 438.342,Z 554.002,A -85,B 0,C 180,E1 -9087.243,E2 -9087.243} C_VEL
LIN {X 0,Y 438.278,Z 555.635,A -85,B 0,C 180,E1 -9089.082,E2 -9089.082} C_VEL
LIN {X 0,Y 438.279,Z 555.855,A -85,B 0,C 180,E1 -9090,E2 -9090} C_VEL
LIN {X 0,Y 438.278,Z 555.638,A -85,B 0,C 180,E1 -9090.919,E2 -9090.919} C_VEL
LIN {X 0,Y 438.342,Z 554.03,A -85,B 0,C 180,E1 -9092.757,E2 -9092.757} C_VEL
LIN {X 0,Y 438.286,Z 552.612,A -85,B 0,C 180,E1 -9093.678,E2 -9093.678} C_VEL
LIN {X 0,Y 438.388,Z 549.651,A -85,B 0,C 180,E1 -9095.059,E2 -9095.059} C_VEL
LIN {X 0,Y 438.449,Z 545.631,A -85,B 0,C 180,E1 -9096.443,E2 -9096.443} C_VEL
LIN {X 0,Y 438.689,Z 539.441,A -85,B 0,C 180,E1 -9098.058,E2 -9098.058} C_VEL
LIN {X 0,Y 439.026,Z 532.689,A -85,B 0,C 180,E1 -9099.444,E2 -9099.444} C_VEL
LIN {X 0,Y 439.439,Z 524.31,A -85,B 0,C 180,E1 -9100.832,E2 -9100.832} C_VEL
LIN {X 0,Y 440.045,Z 515.691,A -85,B 0,C 180,E1 -9101.983,E2 -9101.983} C_VEL
LIN {X 0,Y 440.541,Z 505.993,A -85,B 0,C 180,E1 -9103.048,E2 -9103.048} C_VEL
LIN {X 0,Y 441.184,Z 494.564,A -85,B 0,C 180,E1 -9104.06,E2 -9104.06} C_VEL
LIN {X 0,Y 441.847,Z 482.981,A -85,B 0,C 180,E1 -9104.862,E2 -9104.862} C_VEL
LIN {X 0,Y 442.118,Z 472.29,A -85,B 0,C 180,E1 -9105.442,E2 -9105.442} C_VEL
LIN {X 0,Y 440.256,Z 458.524,A -85,B 0,C 180,E1 -9106.055,E2 -9106.055} C_VEL
LIN {X 0,Y 438.721,Z 448.929,A -85,B 0,C 180,E1 -9106.379,E2 -9106.379} C_VEL
LIN {X 0,Y 438.95,Z 441.049,A -85,B 0,C 180,E1 -9109.648,E2 -9109.648} C_VEL
LIN {X 0,Y 439.217,Z 432.916,A -85,B 0,C 180,E1 -9113.081,E2 -9113.081} C_VEL
LIN {X 0,Y 439.568,Z 425.145,A -85,B 0,C 180,E1 -9116.446,E2 -9116.446} C_VEL
LIN {X 0,Y 439.997,Z 417.86,A -85,B 0,C 180,E1 -9119.68,E2 -9119.68} C_VEL
LIN {X 0,Y 440.44,Z 410.951,A -85,B 0,C 180,E1 -9122.856,E2 -9122.856} C_VEL
LIN {X 0,Y 440.738,Z 405.22,A -85,B 0,C 180,E1 -9125.585,E2 -9125.585} C_VEL
LIN {X 0,Y 440.252,Z 400.616,A -85,B 0,C 180,E1 -9127.916,E2 -9127.916} C_VEL
LIN {X 0,Y 439.427,Z 395.751,A -85,B 0,C 180,E1 -9130.538,E2 -9130.538} C_VEL
LIN {X 0,Y 439.367,Z 395.758,A -85,B 0,C 180,E1 -9133.961,E2 -9133.961} C_VEL
LIN {X 0,Y 439.352,Z 395.757,A -85,B 0,C 180,E1 -9136.54,E2 -9136.54} C_VEL
LIN {X 0,Y 439.382,Z 395.755,A -85,B 0,C 180,E1 -9139.019,E2 -9139.019} C_VEL
LIN {X 0,Y 439.375,Z 395.757,A -85,B 0,C 180,E1 -9141.608,E2 -9141.608} C_VEL
LIN {X 0,Y 439.401,Z 395.753,A -85,B 0,C 180,E1 -9144.844,E2 -9144.844} C_VEL
LIN {X 0,Y 439.373,Z 395.754,A -85,B 0,C 180,E1 -9148.139,E2 -9148.139} C_VEL
LIN {X 0,Y 439.433,Z 395.748,A -85,B 0,C 180,E1 -9151.598,E2 -9151.598} C_VEL
LIN {X 0,Y 439.406,Z 395.751,A -85,B 0,C 180,E1 -9154.415,E2 -9154.415} C_VEL
LIN {X 0,Y 439.365,Z 395.757,A -85,B 0,C 180,E1 -9157.424,E2 -9157.424} C_VEL
LIN {X 0,Y 439.442,Z 395.747,A -85,B 0,C 180,E1 -9160.663,E2 -9160.663} C_VEL
LIN {X 0,Y 439.463,Z 395.743,A -85,B 0,C 180,E1 -9164.224,E2 -9164.224} C_VEL
LIN {X 0,Y 439.484,Z 395.741,A -85,B 0,C 180,E1 -9168.001,E2 -9168.001} C_VEL
LIN {X 0,Y 439.549,Z 395.733,A -85,B 0,C 180,E1 -9171.726,E2 -9171.726} C_VEL
LIN {X 0,Y 439.621,Z 395.726,A -85,B 0,C 180,E1 -9174.496,E2 -9174.496} C_VEL
LIN {X 0,Y 439.634,Z 395.722,A -85,B 0,C 180,E1 -9178.168,E2 -9178.168} C_VEL
LIN {X 0,Y 439.763,Z 395.706,A -85,B 0,C 180,E1 -9180,E2 -9180} C_VEL
LIN {X 0,Y 439.641,Z 395.724,A -85,B 0,C 180,E1 -9182.749,E2 -9182.749} C_VEL
LIN {X 0,Y 439.618,Z 395.726,A -85,B 0,C 180,E1 -9186.425,E2 -9186.425} C_VEL
LIN {X 0,Y 439.5,Z 395.741,A -85,B 0,C 180,E1 -9189.202,E2 -9189.202} C_VEL
LIN {X 0,Y 439.466,Z 395.746,A -85,B 0,C 180,E1 -9192.938,E2 -9192.938} C_VEL
LIN {X 0,Y 439.448,Z 395.746,A -85,B 0,C 180,E1 -9196.349,E2 -9196.349} C_VEL
LIN {X 0,Y 439.403,Z 395.75,A -85,B 0,C 180,E1 -9199.626,E2 -9199.626} C_VEL
LIN {X 0,Y 439.365,Z 395.758,A -85,B 0,C 180,E1 -9202.575,E2 -9202.575} C_VEL
LIN {X 0,Y 439.405,Z 395.75,A -85,B 0,C 180,E1 -9205.585,E2 -9205.585} C_VEL
LIN {X 0,Y 439.418,Z 395.753,A -85,B 0,C 180,E1 -9208.673,E2 -9208.673} C_VEL
LIN {X 0,Y 439.37,Z 395.755,A -85,B 0,C 180,E1 -9212.03,E2 -9212.03} C_VEL
LIN {X 0,Y 439.397,Z 395.753,A -85,B 0,C 180,E1 -9215.341,E2 -9215.341} C_VEL
LIN {X 0,Y 439.378,Z 395.756,A -85,B 0,C 180,E1 -9218.596,E2 -9218.596} C_VEL
LIN {X 0,Y 439.389,Z 395.754,A -85,B 0,C 180,E1 -9221.257,E2 -9221.257} C_VEL
LIN {X 0,Y 439.4,Z 395.753,A -85,B 0,C 180,E1 -9224.729,E2 -9224.729} C_VEL
LIN {X 0,Y 439.397,Z 395.752,A -85,B 0,C 180,E1 -9227.796,E2 -9227.796} C_VEL
LIN {X 0,Y 439.431,Z 395.75,A -85,B 0,C 180,E1 -9230.228,E2 -9230.228} C_VEL
LIN {X 0,Y 439.378,Z 395.754,A -85,B 0,C 180,E1 -9233.713,E2 -9233.713} C_VEL
LIN {X 0,Y 439.374,Z 395.756,A -85,B 0,C 180,E1 -9237.054,E2 -9237.054} C_VEL
LIN {X 0,Y 439.384,Z 395.755,A -85,B 0,C 180,E1 -9240.274,E2 -9240.274} C_VEL
LIN {X 0,Y 439.43,Z 395.747,A -85,B 0,C 180,E1 -9243.396,E2 -9243.396} C_VEL
LIN {X 0,Y 439.389,Z 395.755,A -85,B 0,C 180,E1 -9246.43,E2 -9246.43} C_VEL
LIN {X 0,Y 439.39,Z 395.752,A -85,B 0,C 180,E1 -9249.397,E2 -9249.397} C_VEL
LIN {X 0,Y 439.433,Z 395.749,A -85,B 0,C 180,E1 -9252.309,E2 -9252.309} C_VEL
LIN {X 0,Y 439.45,Z 395.745,A -85,B 0,C 180,E1 -9255.174,E2 -9255.174} C_VEL
LIN {X 0,Y 439.486,Z 395.743,A -85,B 0,C 180,E1 -9258.001,E2 -9258.001} C_VEL
LIN {X 0,Y 439.55,Z 395.733,A -85,B 0,C 180,E1 -9261.726,E2 -9261.726} C_VEL
LIN {X 0,Y 439.623,Z 395.727,A -85,B 0,C 180,E1 -9264.496,E2 -9264.496} C_VEL
LIN {X 0,Y 439.635,Z 395.724,A -85,B 0,C 180,E1 -9268.167,E2 -9268.167} C_VEL
LIN {X 0,Y 439.765,Z 395.708,A -85,B 0,C 180,E1 -9270,E2 -9270} C_VEL
LIN {X 0,Y 439.611,Z 395.724,A -85,B 0,C 180,E1 -9270.983,E2 -9270.983} C_VEL
LIN {X 0,Y 438.904,Z 395.815,A -85,B 0,C 180,E1 -9271.747,E2 -9271.747} C_VEL
LIN {X 0,Y 435.933,Z 396.184,A -85,B 0,C 180,E1 -9272.986,E2 -9272.986} C_VEL
LIN {X 0,Y 433.478,Z 396.491,A -85,B 0,C 180,E1 -9273.987,E2 -9273.987} C_VEL
LIN {X 0,Y 432.496,Z 396.612,A -85,B 0,C 180,E1 -9274.761,E2 -9274.761} C_VEL
LIN {X 0,Y 432.455,Z 396.616,A -85,B 0,C 180,E1 -9275.023,E2 -9275.023} C_VEL
LIN {X 0,Y 432.5,Z 396.613,A -85,B 0,C 180,E1 -9276.531,E2 -9276.531} C_VEL
LIN {X 0,Y 432.113,Z 396.788,A -85,B 0,C 180,E1 -9279.36,E2 -9279.36} C_VEL
LIN {X 0,Y 431.988,Z 400.668,A -85,B 0,C 180,E1 -9282.541,E2 -9282.541} C_VEL
LIN {X 0,Y 431.798,Z 405.244,A -85,B 0,C 180,E1 -9286.2,E2 -9286.2} C_VEL
LIN {X 0,Y 431.641,Z 409.078,A -85,B 0,C 180,E1 -9289.203,E2 -9289.203} C_VEL
LIN {X 0,Y 431.495,Z 414.006,A -85,B 0,C 180,E1 -9293.01,E2 -9293.01} C_VEL
LIN {X 0,Y 431.385,Z 418.65,A -85,B 0,C 180,E1 -9296.461,E2 -9296.461} C_VEL
LIN {X 0,Y 434.374,Z 432.029,A -85,B 0,C 180,E1 -9297.009,E2 -9297.009} C_VEL
LIN {X 0,Y 435.77,Z 439.99,A -85,B 0,C 180,E1 -9297.415,E2 -9297.415} C_VEL
LIN {X 0,Y 435.16,Z 452.44,A -85,B 0,C 180,E1 -9298.124,E2 -9298.124} C_VEL
LIN {X 0,Y 434.509,Z 464.53,A -85,B 0,C 180,E1 -9299.027,E2 -9299.027} C_VEL
LIN {X 0,Y 433.945,Z 474.835,A -85,B 0,C 180,E1 -9300.002,E2 -9300.002} C_VEL
LIN {X 0,Y 433.347,Z 484.397,A -85,B 0,C 180,E1 -9301.12,E2 -9301.12} C_VEL
LIN {X 0,Y 432.75,Z 493.368,A -85,B 0,C 180,E1 -9302.406,E2 -9302.406} C_VEL
LIN {X 0,Y 432.284,Z 501.058,A -85,B 0,C 180,E1 -9303.765,E2 -9303.765} C_VEL
LIN {X 0,Y 431.9,Z 507.253,A -85,B 0,C 180,E1 -9305.12,E2 -9305.12} C_VEL
LIN {X 0,Y 431.607,Z 512.182,A -85,B 0,C 180,E1 -9306.463,E2 -9306.463} C_VEL
LIN {X 0,Y 431.361,Z 517.101,A -85,B 0,C 180,E1 -9308.251,E2 -9308.251} C_VEL
LIN {X 0,Y 431.133,Z 520.349,A -85,B 0,C 180,E1 -9309.99,E2 -9309.99} C_VEL
LIN {X 0,Y 431.086,Z 521.907,A -85,B 0,C 180,E1 -9311.415,E2 -9311.415} C_VEL
LIN {X 0,Y 431.099,Z 522.556,A -85,B 0,C 180,E1 -9313.212,E2 -9313.212} C_VEL
LIN {X 0,Y 431.114,Z 522.125,A -85,B 0,C 180,E1 -9314.505,E2 -9314.505} C_VEL
LIN {X 0,Y 431.163,Z 520.872,A -85,B 0,C 180,E1 -9315.823,E2 -9315.823} C_VEL
LIN {X 0,Y 431.321,Z 518.786,A -85,B 0,C 180,E1 -9317.157,E2 -9317.157} C_VEL
LIN {X 0,Y 431.513,Z 514.651,A -85,B 0,C 180,E1 -9318.942,E2 -9318.942} C_VEL
LIN {X 0,Y 431.862,Z 509.178,A -85,B 0,C 180,E1 -9320.604,E2 -9320.604} C_VEL
LIN {X 0,Y 432.206,Z 502.878,A -85,B 0,C 180,E1 -9322.084,E2 -9322.084} C_VEL
LIN {X 0,Y 432.644,Z 496.208,A -85,B 0,C 180,E1 -9323.347,E2 -9323.347} C_VEL
LIN {X 0,Y 433.29,Z 487.416,A -85,B 0,C 180,E1 -9324.701,E2 -9324.701} C_VEL
LIN {X 0,Y 433.952,Z 477.567,A -85,B 0,C 180,E1 -9325.917,E2 -9325.917} C_VEL
LIN {X 0,Y 434.638,Z 467.12,A -85,B 0,C 180,E1 -9326.96,E2 -9326.96} C_VEL
LIN {X 0,Y 435.233,Z 455.726,A -85,B 0,C 180,E1 -9327.869,E2 -9327.869} C_VEL
LIN {X 0,Y 435.845,Z 444.824,A -85,B 0,C 180,E1 -9328.541,E2 -9328.541} C_VEL
LIN {X 0,Y 435.881,Z 438.58,A -85,B 0,C 180,E1 -9328.865,E2 -9328.865} C_VEL
LIN {X 0,Y 433.094,Z 425.876,A -85,B 0,C 180,E1 -9329.495,E2 -9329.495} C_VEL
LIN {X 0,Y 431.485,Z 419.315,A -85,B 0,C 180,E1 -9329.767,E2 -9329.767} C_VEL
LIN {X 0,Y 431.569,Z 415.373,A -85,B 0,C 180,E1 -9332.872,E2 -9332.872} C_VEL
LIN {X 0,Y 431.791,Z 411.46,A -85,B 0,C 180,E1 -9335.989,E2 -9335.989} C_VEL
LIN {X 0,Y 431.879,Z 407.774,A -85,B 0,C 180,E1 -9339.022,E2 -9339.022} C_VEL
LIN {X 0,Y 432.048,Z 404.193,A -85,B 0,C 180,E1 -9341.997,E2 -9341.997} C_VEL
LIN {X 0,Y 432.174,Z 400.785,A -85,B 0,C 180,E1 -9344.919,E2 -9344.919} C_VEL
LIN {X 0,Y 432.37,Z 397.495,A -85,B 0,C 180,E1 -9347.801,E2 -9347.801} C_VEL
LIN {X 0,Y 432.312,Z 396.638,A -85,B 0,C 180,E1 -9348.751,E2 -9348.751} C_VEL
LIN {X 0,Y 432.581,Z 396.605,A -85,B 0,C 180,E1 -9352.321,E2 -9352.321} C_VEL
LIN {X 0,Y 432.594,Z 396.603,A -85,B 0,C 180,E1 -9354.406,E2 -9354.406} C_VEL
LIN {X 0,Y 432.602,Z 396.602,A -85,B 0,C 180,E1 -9358.138,E2 -9358.138} C_VEL
LIN {X 0,Y 432.731,Z 396.584,A -85,B 0,C 180,E1 -9360,E2 -9360} C_VEL
LIN {X 0,Y 432.601,Z 396.6,A -85,B 0,C 180,E1 -9362.794,E2 -9362.794} C_VEL
LIN {X 0,Y 432.569,Z 396.604,A -85,B 0,C 180,E1 -9366.53,E2 -9366.53} C_VEL
LIN {X 0,Y 432.439,Z 396.62,A -85,B 0,C 180,E1 -9369.353,E2 -9369.353} C_VEL
LIN {X 0,Y 432.426,Z 396.622,A -85,B 0,C 180,E1 -9372.804,E2 -9372.804} C_VEL
LIN {X 0,Y 432.408,Z 396.625,A -85,B 0,C 180,E1 -9376.479,E2 -9376.479} C_VEL
LIN {X 0,Y 432.335,Z 396.632,A -85,B 0,C 180,E1 -9379.961,E2 -9379.961} C_VEL
LIN {X 0,Y 432.316,Z 396.636,A -85,B 0,C 180,E1 -9382.965,E2 -9382.965} C_VEL
LIN {X 0,Y 432.361,Z 396.63,A -85,B 0,C 180,E1 -9386.033,E2 -9386.033} C_VEL
LIN {X 0,Y 432.349,Z 396.631,A -85,B 0,C 180,E1 -9389.187,E2 -9389.187} C_VEL
LIN {X 0,Y 432.322,Z 396.635,A -85,B 0,C 180,E1 -9392.294,E2 -9392.294} C_VEL
LIN {X 0,Y 432.338,Z 396.634,A -85,B 0,C 180,E1 -9394.677,E2 -9394.677} C_VEL
LIN {X 0,Y 432.351,Z 396.634,A -85,B 0,C 180,E1 -9398.149,E2 -9398.149} C_VEL
LIN {X 0,Y 432.364,Z 396.632,A -85,B 0,C 180,E1 -9401.608,E2 -9401.608} C_VEL
LIN {X 0,Y 432.331,Z 396.635,A -85,B 0,C 180,E1 -9404.348,E2 -9404.348} C_VEL
LIN {X 0,Y 432.319,Z 396.635,A -85,B 0,C 180,E1 -9407.016,E2 -9407.016} C_VEL
LIN {X 0,Y 432.368,Z 396.745,A -85,B 0,C 180,E1 -9408.567,E2 -9408.567} C_VEL
LIN {X 0,Y 433.35,Z 402.312,A -85,B 0,C 180,E1 -9411.956,E2 -9411.956} C_VEL
LIN {X 0,Y 433.741,Z 406.569,A -85,B 0,C 180,E1 -9414.317,E2 -9414.317} C_VEL
LIN {X 0,Y 433.55,Z 410.919,A -85,B 0,C 180,E1 -9416.555,E2 -9416.555} C_VEL
LIN {X 0,Y 432.998,Z 417.564,A -85,B 0,C 180,E1 -9419.791,E2 -9419.791} C_VEL
LIN {X 0,Y 432.556,Z 424.323,A -85,B 0,C 180,E1 -9422.94,E2 -9422.94} C_VEL
LIN {X 0,Y 432.226,Z 431.141,A -85,B 0,C 180,E1 -9426.015,E2 -9426.015} C_VEL
LIN {X 0,Y 431.936,Z 438.066,A -85,B 0,C 180,E1 -9429.026,E2 -9429.026} C_VEL
LIN {X 0,Y 431.656,Z 446.179,A -85,B 0,C 180,E1 -9432.47,E2 -9432.47} C_VEL
LIN {X 0,Y 431.637,Z 447.995,A -85,B 0,C 180,E1 -9433.229,E2 -9433.229} C_VEL
LIN {X 0,Y 434.012,Z 462.523,A -85,B 0,C 180,E1 -9433.783,E2 -9433.783} C_VEL
LIN {X 0,Y 435.427,Z 474.28,A -85,B 0,C 180,E1 -9434.375,E2 -9434.375} C_VEL
LIN {X 0,Y 434.802,Z 486.947,A -85,B 0,C 180,E1 -9435.132,E2 -9435.132} C_VEL
LIN {X 0,Y 434.041,Z 498.675,A -85,B 0,C 180,E1 -9436.045,E2 -9436.045} C_VEL
LIN {X 0,Y 433.426,Z 509.537,A -85,B 0,C 180,E1 -9437.118,E2 -9437.118} C_VEL
LIN {X 0,Y 432.84,Z 519.177,A -85,B 0,C 180,E1 -9438.29,E2 -9438.29} C_VEL
LIN {X 0,Y 432.258,Z 527.095,A -85,B 0,C 180,E1 -9439.461,E2 -9439.461} C_VEL
LIN {X 0,Y 431.834,Z 534.848,A -85,B 0,C 180,E1 -9440.87,E2 -9440.87} C_VEL
LIN {X 0,Y 431.5,Z 542.014,A -85,B 0,C 180,E1 -9442.514,E2 -9442.514} C_VEL
LIN {X 0,Y 431.286,Z 547.085,A -85,B 0,C 180,E1 -9444.017,E2 -9444.017} C_VEL
LIN {X 0,Y 431.275,Z 550.439,A -85,B 0,C 180,E1 -9445.327,E2 -9445.327} C_VEL
LIN {X 0,Y 431.193,Z 552.32,A -85,B 0,C 180,E1 -9446.262,E2 -9446.262} C_VEL
LIN {X 0,Y 431.238,Z 553.735,A -85,B 0,C 180,E1 -9447.198,E2 -9447.198} C_VEL
LIN {X 0,Y 431.219,Z 554.747,A -85,B 0,C 180,E1 -9448.132,E2 -9448.132} C_VEL
LIN {X 0,Y 431.193,Z 555.366,A -85,B 0,C 180,E1 -9449.066,E2 -9449.066} C_VEL
LIN {X 0,Y 431.192,Z 555.582,A -85,B 0,C 180,E1 -9450,E2 -9450} C_VEL
LIN {X 0,Y 431.219,Z 554.751,A -85,B 0,C 180,E1 -9451.868,E2 -9451.868} C_VEL
LIN {X 0,Y 431.253,Z 553.748,A -85,B 0,C 180,E1 -9452.803,E2 -9452.803} C_VEL
LIN {X 0,Y 431.193,Z 552.324,A -85,B 0,C 180,E1 -9453.738,E2 -9453.738} C_VEL
LIN {X 0,Y 431.299,Z 549.356,A -85,B 0,C 180,E1 -9455.142,E2 -9455.142} C_VEL
LIN {X 0,Y 431.377,Z 545.328,A -85,B 0,C 180,E1 -9456.549,E2 -9456.549} C_VEL
LIN {X 0,Y 431.62,Z 539.124,A -85,B 0,C 180,E1 -9458.191,E2 -9458.191} C_VEL
LIN {X 0,Y 431.985,Z 532.361,A -85,B 0,C 180,E1 -9459.6,E2 -9459.6} C_VEL
LIN {X 0,Y 432.434,Z 523.965,A -85,B 0,C 180,E1 -9461.009,E2 -9461.009} C_VEL
LIN {X 0,Y 433.053,Z 515.325,A -85,B 0,C 180,E1 -9462.18,E2 -9462.18} C_VEL
LIN {X 0,Y 433.62,Z 505.084,A -85,B 0,C 180,E1 -9463.314,E2 -9463.314} C_VEL
LIN {X 0,Y 434.269,Z 494.158,A -85,B 0,C 180,E1 -9464.288,E2 -9464.288} C_VEL
LIN {X 0,Y 434.956,Z 482.523,A -85,B 0,C 180,E1 -9465.103,E2 -9465.103} C_VEL
LIN {X 0,Y 435.19,Z 473.029,A -85,B 0,C 180,E1 -9465.634,E2 -9465.634} C_VEL
LIN {X 0,Y 433.504,Z 460.129,A -85,B 0,C 180,E1 -9466.239,E2 -9466.239} C_VEL
LIN {X 0,Y 431.65,Z 448.696,A -85,B 0,C 180,E1 -9466.642,E2 -9466.642} C_VEL
LIN {X 0,Y 431.896,Z 440.789,A -85,B 0,C 180,E1 -9469.982,E2 -9469.982} C_VEL
LIN {X 0,Y 432.153,Z 433.848,A -85,B 0,C 180,E1 -9472.974,E2 -9472.974} C_VEL
LIN {X 0,Y 432.448,Z 426.892,A -85,B 0,C 180,E1 -9476.027,E2 -9476.027} C_VEL
LIN {X 0,Y 432.875,Z 419.978,A -85,B 0,C 180,E1 -9479.148,E2 -9479.148} C_VEL
LIN {X 0,Y 433.34,Z 412.752,A -85,B 0,C 180,E1 -9482.504,E2 -9482.504} C_VEL
LIN {X 0,Y 433.689,Z 407.326,A -85,B 0,C 180,E1 -9485.12,E2 -9485.12} C_VEL
LIN {X 0,Y 433.42,Z 402.841,A -85,B 0,C 180,E1 -9487.387,E2 -9487.387} C_VEL
LIN {X 0,Y 432.403,Z 396.648,A -85,B 0,C 180,E1 -9490.724,E2 -9490.724} C_VEL
LIN {X 0,Y 432.335,Z 396.634,A -85,B 0,C 180,E1 -9494.347,E2 -9494.347} C_VEL
LIN {X 0,Y 432.321,Z 396.635,A -85,B 0,C 180,E1 -9497.016,E2 -9497.016} C_VEL
LIN {X 0,Y 432.334,Z 396.631,A -85,B 0,C 180,E1 -9499.821,E2 -9499.821} C_VEL
LIN {X 0,Y 432.308,Z 396.637,A -85,B 0,C 180,E1 -9503.022,E2 -9503.022} C_VEL
LIN {X 0,Y 432.36,Z 396.627,A -85,B 0,C 180,E1 -9505.996,E2 -9505.996} C_VEL
LIN {X 0,Y 432.348,Z 396.631,A -85,B 0,C 180,E1 -9509.49,E2 -9509.49} C_VEL
LIN {X 0,Y 432.392,Z 396.627,A -85,B 0,C 180,E1 -9512.928,E2 -9512.928} C_VEL
LIN {X 0,Y 432.372,Z 396.627,A -85,B 0,C 180,E1 -9516.023,E2 -9516.023} C_VEL
LIN {X 0,Y 432.351,Z 396.632,A -85,B 0,C 180,E1 -9519.046,E2 -9519.046} C_VEL
LIN {X 0,Y 432.378,Z 396.626,A -85,B 0,C 180,E1 -9522.011,E2 -9522.011} C_VEL
LIN {X 0,Y 432.396,Z 396.626,A -85,B 0,C 180,E1 -9524.926,E2 -9524.926} C_VEL
LIN {X 0,Y 432.46,Z 396.616,A -85,B 0,C 180,E1 -9527.803,E2 -9527.803} C_VEL
LIN {X 0,Y 432.493,Z 396.613,A -85,B 0,C 180,E1 -9531.59,E2 -9531.59} C_VEL
LIN {X 0,Y 432.597,Z 396.6,A -85,B 0,C 180,E1 -9534.406,E2 -9534.406} C_VEL
LIN {X 0,Y 432.604,Z 396.598,A -85,B 0,C 180,E1 -9538.138,E2 -9538.138} C_VEL
LIN {X 0,Y 432.732,Z 396.582,A -85,B 0,C 180,E1 -9540,E2 -9540} C_VEL
LIN {X 0,Y 432.592,Z 396.602,A -85,B 0,C 180,E1 -9542.794,E2 -9542.794} C_VEL
LIN {X 0,Y 432.573,Z 396.604,A -85,B 0,C 180,E1 -9546.53,E2 -9546.53} C_VEL
LIN {X 0,Y 432.443,Z 396.62,A -85,B 0,C 180,E1 -9549.353,E2 -9549.353} C_VEL
LIN {X 0,Y 432.431,Z 396.622,A -85,B 0,C 180,E1 -9552.803,E2 -9552.803} C_VEL
LIN {X 0,Y 432.413,Z 396.623,A -85,B 0,C 180,E1 -9556.479,E2 -9556.479} C_VEL
LIN {X 0,Y 432.339,Z 396.63,A -85,B 0,C 180,E1 -9559.96,E2 -9559.96} C_VEL
LIN {X 0,Y 432.319,Z 396.635,A -85,B 0,C 180,E1 -9562.964,E2 -9562.964} C_VEL
LIN {X 0,Y 432.364,Z 396.627,A -85,B 0,C 180,E1 -9566.032,E2 -9566.032} C_VEL
LIN {X 0,Y 432.343,Z 396.631,A -85,B 0,C 180,E1 -9569.187,E2 -9569.187} C_VEL
LIN {X 0,Y 432.323,Z 396.636,A -85,B 0,C 180,E1 -9572.443,E2 -9572.443} C_VEL
LIN {X 0,Y 432.346,Z 396.63,A -85,B 0,C 180,E1 -9575.632,E2 -9575.632} C_VEL
LIN {X 0,Y 432.341,Z 396.633,A -85,B 0,C 180,E1 -9578.714,E2 -9578.714} C_VEL
LIN {X 0,Y 432.334,Z 396.631,A -85,B 0,C 180,E1 -9581.797,E2 -9581.797} C_VEL
LIN {X 0,Y 432.334,Z 396.634,A -85,B 0,C 180,E1 -9584.347,E2 -9584.347} C_VEL
LIN {X 0,Y 432.321,Z 396.634,A -85,B 0,C 180,E1 -9587.016,E2 -9587.016} C_VEL
LIN {X 0,Y 432.337,Z 396.63,A -85,B 0,C 180,E1 -9589.82,E2 -9589.82} C_VEL
LIN {X 0,Y 432.317,Z 396.635,A -85,B 0,C 180,E1 -9593.023,E2 -9593.023} C_VEL
LIN {X 0,Y 432.361,Z 396.628,A -85,B 0,C 180,E1 -9595.996,E2 -9595.996} C_VEL
LIN {X 0,Y 432.349,Z 396.629,A -85,B 0,C 180,E1 -9599.49,E2 -9599.49} C_VEL
LIN {X 0,Y 432.393,Z 396.626,A -85,B 0,C 180,E1 -9602.928,E2 -9602.928} C_VEL
LIN {X 0,Y 432.373,Z 396.629,A -85,B 0,C 180,E1 -9606.023,E2 -9606.023} C_VEL
LIN {X 0,Y 432.352,Z 396.63,A -85,B 0,C 180,E1 -9609.046,E2 -9609.046} C_VEL
LIN {X 0,Y 432.379,Z 396.628,A -85,B 0,C 180,E1 -9612.011,E2 -9612.011} C_VEL
LIN {X 0,Y 432.398,Z 396.625,A -85,B 0,C 180,E1 -9614.926,E2 -9614.926} C_VEL
LIN {X 0,Y 432.461,Z 396.617,A -85,B 0,C 180,E1 -9617.803,E2 -9617.803} C_VEL
LIN {X 0,Y 432.494,Z 396.612,A -85,B 0,C 180,E1 -9621.59,E2 -9621.59} C_VEL
LIN {X 0,Y 432.6,Z 396.601,A -85,B 0,C 180,E1 -9624.406,E2 -9624.406} C_VEL
LIN {X 0,Y 432.605,Z 396.6,A -85,B 0,C 180,E1 -9628.138,E2 -9628.138} C_VEL
LIN {X 0,Y 432.734,Z 396.584,A -85,B 0,C 180,E1 -9630,E2 -9630} C_VEL
LIN {X 0,Y 432.607,Z 396.599,A -85,B 0,C 180,E1 -9632.793,E2 -9632.793} C_VEL
LIN {X 0,Y 432.455,Z 396.616,A -85,B 0,C 180,E1 -9635.023,E2 -9635.023} C_VEL
LIN {X 0,Y 431.869,Z 396.691,A -85,B 0,C 180,E1 -9635.801,E2 -9635.801} C_VEL
LIN {X 0,Y 428.94,Z 397.053,A -85,B 0,C 180,E1 -9637.062,E2 -9637.062} C_VEL
LIN {X 0,Y 426.366,Z 397.378,A -85,B 0,C 180,E1 -9638.079,E2 -9638.079} C_VEL
LIN {X 0,Y 425.214,Z 397.618,A -85,B 0,C 180,E1 -9638.868,E2 -9638.868} C_VEL
LIN {X 0,Y 425.1,Z 397.698,A -85,B 0,C 180,E1 -9639.135,E2 -9639.135} C_VEL
LIN {X 0,Y 425.066,Z 397.812,A -85,B 0,C 180,E1 -9639.516,E2 -9639.516} C_VEL
LIN {X 0,Y 424.93,Z 401.573,A -85,B 0,C 180,E1 -9642.627,E2 -9642.627} C_VEL
LIN {X 0,Y 424.728,Z 406.147,A -85,B 0,C 180,E1 -9646.337,E2 -9646.337} C_VEL
LIN {X 0,Y 424.566,Z 409.96,A -85,B 0,C 180,E1 -9649.344,E2 -9649.344} C_VEL
LIN {X 0,Y 424.431,Z 413.895,A -85,B 0,C 180,E1 -9652.386,E2 -9652.386} C_VEL
LIN {X 0,Y 424.309,Z 417.933,A -85,B 0,C 180,E1 -9655.508,E2 -9655.508} C_VEL
LIN {X 0,Y 424.344,Z 419.001,A -85,B 0,C 180,E1 -9656.198,E2 -9656.198} C_VEL
LIN {X 0,Y 427.407,Z 432.554,A -85,B 0,C 180,E1 -9656.77,E2 -9656.77} C_VEL
LIN {X 0,Y 428.858,Z 440.429,A -85,B 0,C 180,E1 -9657.184,E2 -9657.184} C_VEL
LIN {X 0,Y 428.315,Z 452.138,A -85,B 0,C 180,E1 -9657.859,E2 -9657.859} C_VEL
LIN {X 0,Y 427.618,Z 463.825,A -85,B 0,C 180,E1 -9658.732,E2 -9658.732} C_VEL
LIN {X 0,Y 427.057,Z 474.283,A -85,B 0,C 180,E1 -9659.719,E2 -9659.719} C_VEL
LIN {X 0,Y 426.379,Z 484.412,A -85,B 0,C 180,E1 -9660.905,E2 -9660.905} C_VEL
LIN {X 0,Y 425.778,Z 493.653,A -85,B 0,C 180,E1 -9662.25,E2 -9662.25} C_VEL
LIN {X 0,Y 425.269,Z 501.266,A -85,B 0,C 180,E1 -9663.615,E2 -9663.615} C_VEL
LIN {X 0,Y 424.828,Z 507.863,A -85,B 0,C 180,E1 -9665.09,E2 -9665.09} C_VEL
LIN {X 0,Y 424.499,Z 513.114,A -85,B 0,C 180,E1 -9666.584,E2 -9666.584} C_VEL
LIN {X 0,Y 424.273,Z 517.68,A -85,B 0,C 180,E1 -9668.322,E2 -9668.322} C_VEL
LIN {X 0,Y 424.167,Z 519.088,A -85,B 0,C 180,E1 -9669.021,E2 -9669.021} C_VEL
LIN {X 0,Y 424.036,Z 521.094,A -85,B 0,C 180,E1 -9670.323,E2 -9670.323} C_VEL
LIN {X 0,Y 423.987,Z 522.419,A -85,B 0,C 180,E1 -9671.762,E2 -9671.762} C_VEL
LIN {X 0,Y 424.004,Z 522.838,A -85,B 0,C 180,E1 -9673.171,E2 -9673.171} C_VEL
LIN {X 0,Y 424.02,Z 522.398,A -85,B 0,C 180,E1 -9674.544,E2 -9674.544} C_VEL
LIN {X 0,Y 424.076,Z 521.139,A -85,B 0,C 180,E1 -9675.889,E2 -9675.889} C_VEL
LIN {X 0,Y 424.236,Z 519.102,A -85,B 0,C 180,E1 -9677.218,E2 -9677.218} C_VEL
LIN {X 0,Y 424.373,Z 516.324,A -85,B 0,C 180,E1 -9678.514,E2 -9678.514} C_VEL
LIN {X 0,Y 424.671,Z 511.679,A -85,B 0,C 180,E1 -9680.113,E2 -9680.113} C_VEL
LIN {X 0,Y 425.05,Z 505.714,A -85,B 0,C 180,E1 -9681.681,E2 -9681.681} C_VEL
LIN {X 0,Y 425.499,Z 499.373,A -85,B 0,C 180,E1 -9683.007,E2 -9683.007} C_VEL
LIN {X 0,Y 426.041,Z 491.464,A -85,B 0,C 180,E1 -9684.355,E2 -9684.355} C_VEL
LIN {X 0,Y 426.786,Z 481.547,A -85,B 0,C 180,E1 -9685.707,E2 -9685.707} C_VEL
LIN {X 0,Y 427.473,Z 471.905,A -85,B 0,C 180,E1 -9686.773,E2 -9686.773} C_VEL
LIN {X 0,Y 428.164,Z 460.815,A -85,B 0,C 180,E1 -9687.76,E2 -9687.76} C_VEL
LIN {X 0,Y 428.756,Z 449.221,A -85,B 0,C 180,E1 -9688.569,E2 -9688.569} C_VEL
LIN {X 0,Y 429.067,Z 439.767,A -85,B 0,C 180,E1 -9689.092,E2 -9689.092} C_VEL
LIN {X 0,Y 426.189,Z 426.635,A -85,B 0,C 180,E1 -9689.771,E2 -9689.771} C_VEL
LIN {X 0,Y 424.432,Z 419.595,A -85,B 0,C 180,E1 -9690.089,E2 -9690.089} C_VEL
LIN {X 0,Y 424.558,Z 415.38,A -85,B 0,C 180,E1 -9693.452,E2 -9693.452} C_VEL
LIN {X 0,Y 424.723,Z 411.523,A -85,B 0,C 180,E1 -9696.601,E2 -9696.601} C_VEL
LIN {X 0,Y 424.868,Z 407.83,A -85,B 0,C 180,E1 -9699.673,E2 -9699.673} C_VEL
LIN {X 0,Y 425.038,Z 404.293,A -85,B 0,C 180,E1 -9702.685,E2 -9702.685} C_VEL
LIN {X 0,Y 425.194,Z 400.932,A -85,B 0,C 180,E1 -9705.645,E2 -9705.645} C_VEL
LIN {X 0,Y 425.356,Z 398.729,A -85,B 0,C 180,E1 -9707.597,E2 -9707.597} C_VEL
LIN {X 0,Y 425.272,Z 397.695,A -85,B 0,C 180,E1 -9708.562,E2 -9708.562} C_VEL
LIN {X 0,Y 425.437,Z 397.497,A -85,B 0,C 180,E1 -9711.45,E2 -9711.45} C_VEL
LIN {X 0,Y 425.55,Z 397.48,A -85,B 0,C 180,E1 -9714.313,E2 -9714.313} C_VEL
LIN {X 0,Y 425.572,Z 397.477,A -85,B 0,C 180,E1 -9718.107,E2 -9718.107} C_VEL
LIN {X 0,Y 425.7,Z 397.46,A -85,B 0,C 180,E1 -9720,E2 -9720} C_VEL
LIN {X 0,Y 425.553,Z 397.479,A -85,B 0,C 180,E1 -9722.84,E2 -9722.84} C_VEL
LIN {X 0,Y 425.527,Z 397.482,A -85,B 0,C 180,E1 -9726.639,E2 -9726.639} C_VEL
LIN {X 0,Y 425.397,Z 397.497,A -85,B 0,C 180,E1 -9729.51,E2 -9729.51} C_VEL
LIN {X 0,Y 425.389,Z 397.499,A -85,B 0,C 180,E1 -9732.904,E2 -9732.904} C_VEL
LIN {X 0,Y 425.357,Z 397.503,A -85,B 0,C 180,E1 -9736.605,E2 -9736.605} C_VEL
LIN {X 0,Y 425.325,Z 397.506,A -85,B 0,C 180,E1 -9739.636,E2 -9739.636} C_VEL
LIN {X 0,Y 425.303,Z 397.51,A -85,B 0,C 180,E1 -9743.365,E2 -9743.365} C_VEL
LIN {X 0,Y 425.345,Z 397.505,A -85,B 0,C 180,E1 -9746.845,E2 -9746.845} C_VEL
LIN {X 0,Y 425.315,Z 397.508,A -85,B 0,C 180,E1 -9749.718,E2 -9749.718} C_VEL
LIN {X 0,Y 425.279,Z 397.514,A -85,B 0,C 180,E1 -9753.048,E2 -9753.048} C_VEL
LIN {X 0,Y 425.282,Z 397.514,A -85,B 0,C 180,E1 -9755.93,E2 -9755.93} C_VEL
LIN {X 0,Y 425.311,Z 397.511,A -85,B 0,C 180,E1 -9759.047,E2 -9759.047} C_VEL
LIN {X 0,Y 425.313,Z 397.51,A -85,B 0,C 180,E1 -9761.963,E2 -9761.963} C_VEL
LIN {X 0,Y 425.283,Z 397.513,A -85,B 0,C 180,E1 -9765.284,E2 -9765.284} C_VEL
LIN {X 0,Y 425.367,Z 397.655,A -85,B 0,C 180,E1 -9768.238,E2 -9768.238} C_VEL
LIN {X 0,Y 426.156,Z 402.379,A -85,B 0,C 180,E1 -9771.195,E2 -9771.195} C_VEL
LIN {X 0,Y 426.718,Z 406.879,A -85,B 0,C 180,E1 -9773.806,E2 -9773.806} C_VEL
LIN {X 0,Y 426.646,Z 410.875,A -85,B 0,C 180,E1 -9775.94,E2 -9775.94} C_VEL
LIN {X 0,Y 426.035,Z 417.45,A -85,B 0,C 180,E1 -9779.245,E2 -9779.245} C_VEL
LIN {X 0,Y 425.624,Z 423.039,A -85,B 0,C 180,E1 -9781.928,E2 -9781.928} C_VEL
LIN {X 0,Y 425.251,Z 430.464,A -85,B 0,C 180,E1 -9785.364,E2 -9785.364} C_VEL
LIN {X 0,Y 424.929,Z 437.857,A -85,B 0,C 180,E1 -9788.663,E2 -9788.663} C_VEL
LIN {X 0,Y 424.584,Z 445.951,A -85,B 0,C 180,E1 -9792.169,E2 -9792.169} C_VEL
LIN {X 0,Y 424.583,Z 447.707,A -85,B 0,C 180,E1 -9792.925,E2 -9792.925} C_VEL
LIN {X 0,Y 427.06,Z 462.489,A -85,B 0,C 180,E1 -9793.508,E2 -9793.508} C_VEL
LIN {X 0,Y 428.545,Z 475.338,A -85,B 0,C 180,E1 -9794.179,E2 -9794.179} C_VEL
LIN {X 0,Y 427.921,Z 486.835,A -85,B 0,C 180,E1 -9794.887,E2 -9794.887} C_VEL
LIN {X 0,Y 427.131,Z 498.65,A -85,B 0,C 180,E1 -9795.827,E2 -9795.827} C_VEL
LIN {X 0,Y 426.444,Z 509.353,A -85,B 0,C 180,E1 -9796.903,E2 -9796.903} C_VEL
LIN {X 0,Y 425.853,Z 518.978,A -85,B 0,C 180,E1 -9798.095,E2 -9798.095} C_VEL
LIN {X 0,Y 425.137,Z 528.265,A -85,B 0,C 180,E1 -9799.523,E2 -9799.523} C_VEL
LIN {X 0,Y 424.728,Z 535.749,A -85,B 0,C 180,E1 -9800.956,E2 -9800.956} C_VEL
LIN {X 0,Y 424.418,Z 541.77,A -85,B 0,C 180,E1 -9802.388,E2 -9802.388} C_VEL
LIN {X 0,Y 424.244,Z 546.17,A -85,B 0,C 180,E1 -9803.699,E2 -9803.699} C_VEL
LIN {X 0,Y 424.204,Z 550.18,A -85,B 0,C 180,E1 -9805.249,E2 -9805.249} C_VEL
LIN {X 0,Y 424.104,Z 552.055,A -85,B 0,C 180,E1 -9806.2,E2 -9806.2} C_VEL
LIN {X 0,Y 424.135,Z 553.469,A -85,B 0,C 180,E1 -9807.151,E2 -9807.151} C_VEL
LIN {X 0,Y 424.144,Z 554.48,A -85,B 0,C 180,E1 -9808.101,E2 -9808.101} C_VEL
LIN {X 0,Y 424.111,Z 555.098,A -85,B 0,C 180,E1 -9809.051,E2 -9809.051} C_VEL
LIN {X 0,Y 424.108,Z 555.309,A -85,B 0,C 180,E1 -9810,E2 -9810} C_VEL
LIN {X 0,Y 424.144,Z 554.473,A -85,B 0,C 180,E1 -9811.899,E2 -9811.899} C_VEL
LIN {X 0,Y 424.15,Z 553.466,A -85,B 0,C 180,E1 -9812.85,E2 -9812.85} C_VEL
LIN {X 0,Y 424.104,Z 552.036,A -85,B 0,C 180,E1 -9813.801,E2 -9813.801} C_VEL
LIN {X 0,Y 424.212,Z 549.061,A -85,B 0,C 180,E1 -9815.228,E2 -9815.228} C_VEL
LIN {X 0,Y 424.301,Z 545.024,A -85,B 0,C 180,E1 -9816.659,E2 -9816.659} C_VEL
LIN {X 0,Y 424.551,Z 538.807,A -85,B 0,C 180,E1 -9818.329,E2 -9818.329} C_VEL
LIN {X 0,Y 424.938,Z 532.032,A -85,B 0,C 180,E1 -9819.76,E2 -9819.76} C_VEL
LIN {X 0,Y 425.441,Z 523.618,A -85,B 0,C 180,E1 -9821.193,E2 -9821.193} C_VEL
LIN {X 0,Y 426.07,Z 514.952,A -85,B 0,C 180,E1 -9822.383,E2 -9822.383} C_VEL
LIN {X 0,Y 426.684,Z 504.468,A -85,B 0,C 180,E1 -9823.556,E2 -9823.556} C_VEL
LIN {X 0,Y 427.35,Z 493.721,A -85,B 0,C 180,E1 -9824.525,E2 -9824.525} C_VEL
LIN {X 0,Y 428.093,Z 482.017,A -85,B 0,C 180,E1 -9825.351,E2 -9825.351} C_VEL
LIN {X 0,Y 428.367,Z 474.738,A -85,B 0,C 180,E1 -9825.768,E2 -9825.768} C_VEL
LIN {X 0,Y 426.7,Z 461.578,A -85,B 0,C 180,E1 -9826.428,E2 -9826.428} C_VEL
LIN {X 0,Y 424.587,Z 448.431,A -85,B 0,C 180,E1 -9826.916,E2 -9826.916} C_VEL
LIN {X 0,Y 424.837,Z 440.542,A -85,B 0,C 180,E1 -9830.329,E2 -9830.329} C_VEL
LIN {X 0,Y 425.127,Z 433.596,A -85,B 0,C 180,E1 -9833.376,E2 -9833.376} C_VEL
LIN {X 0,Y 425.506,Z 425.807,A -85,B 0,C 180,E1 -9836.886,E2 -9836.886} C_VEL
LIN {X 0,Y 425.933,Z 419.768,A -85,B 0,C 180,E1 -9839.67,E2 -9839.67} C_VEL
LIN {X 0,Y 426.372,Z 412.875,A -85,B 0,C 180,E1 -9842.953,E2 -9842.953} C_VEL
LIN {X 0,Y 426.686,Z 408.278,A -85,B 0,C 180,E1 -9845.204,E2 -9845.204} C_VEL
LIN {X 0,Y 426.353,Z 403.46,A -85,B 0,C 180,E1 -9847.699,E2 -9847.699} C_VEL
LIN {X 0,Y 425.372,Z 397.605,A -85,B 0,C 180,E1 -9850.918,E2 -9850.918} C_VEL
LIN {X 0,Y 425.286,Z 397.511,A -85,B 0,C 180,E1 -9854.717,E2 -9854.717} C_VEL
LIN {X 0,Y 425.291,Z 397.509,A -85,B 0,C 180,E1 -9858.042,E2 -9858.042} C_VEL
LIN {X 0,Y 425.303,Z 397.51,A -85,B 0,C 180,E1 -9861.102,E2 -9861.102} C_VEL
LIN {X 0,Y 425.301,Z 397.509,A -85,B 0,C 180,E1 -9864.664,E2 -9864.664} C_VEL
LIN {X 0,Y 425.265,Z 397.511,A -85,B 0,C 180,E1 -9868.073,E2 -9868.073} C_VEL
LIN {X 0,Y 425.332,Z 397.506,A -85,B 0,C 180,E1 -9871.368,E2 -9871.368} C_VEL
LIN {X 0,Y 425.296,Z 397.508,A -85,B 0,C 180,E1 -9874.555,E2 -9874.555} C_VEL
LIN {X 0,Y 425.289,Z 397.509,A -85,B 0,C 180,E1 -9877.661,E2 -9877.661} C_VEL
LIN {X 0,Y 425.363,Z 397.501,A -85,B 0,C 180,E1 -9880.704,E2 -9880.704} C_VEL
LIN {X 0,Y 425.389,Z 397.496,A -85,B 0,C 180,E1 -9883.688,E2 -9883.688} C_VEL
LIN {X 0,Y 425.413,Z 397.495,A -85,B 0,C 180,E1 -9887.598,E2 -9887.598} C_VEL
LIN {X 0,Y 425.443,Z 397.492,A -85,B 0,C 180,E1 -9891.45,E2 -9891.45} C_VEL
LIN {X 0,Y 425.554,Z 397.477,A -85,B 0,C 180,E1 -9894.313,E2 -9894.313} C_VEL
LIN {X 0,Y 425.573,Z 397.473,A -85,B 0,C 180,E1 -9898.107,E2 -9898.107} C_VEL
LIN {X 0,Y 425.702,Z 397.457,A -85,B 0,C 180,E1 -9900,E2 -9900} C_VEL
LIN {X 0,Y 425.546,Z 397.479,A -85,B 0,C 180,E1 -9902.84,E2 -9902.84} C_VEL
LIN {X 0,Y 425.531,Z 397.481,A -85,B 0,C 180,E1 -9906.639,E2 -9906.639} C_VEL
LIN {X 0,Y 425.401,Z 397.495,A -85,B 0,C 180,E1 -9909.509,E2 -9909.509} C_VEL
LIN {X 0,Y 425.394,Z 397.499,A -85,B 0,C 180,E1 -9912.904,E2 -9912.904} C_VEL
LIN {X 0,Y 425.362,Z 397.502,A -85,B 0,C 180,E1 -9916.605,E2 -9916.605} C_VEL
LIN {X 0,Y 425.329,Z 397.503,A -85,B 0,C 180,E1 -9919.636,E2 -9919.636} C_VEL
LIN {X 0,Y 425.307,Z 397.508,A -85,B 0,C 180,E1 -9923.365,E2 -9923.365} C_VEL
LIN {X 0,Y 425.348,Z 397.504,A -85,B 0,C 180,E1 -9926.844,E2 -9926.844} C_VEL
LIN {X 0,Y 425.291,Z 397.508,A -85,B 0,C 180,E1 -9929.72,E2 -9929.72} C_VEL
LIN {X 0,Y 425.283,Z 397.512,A -85,B 0,C 180,E1 -9933.048,E2 -9933.048} C_VEL
LIN {X 0,Y 425.284,Z 397.51,A -85,B 0,C 180,E1 -9935.929,E2 -9935.929} C_VEL
LIN {X 0,Y 425.288,Z 397.512,A -85,B 0,C 180,E1 -9939.042,E2 -9939.042} C_VEL
LIN {X 0,Y 425.29,Z 397.509,A -85,B 0,C 180,E1 -9941.958,E2 -9941.958} C_VEL
LIN {X 0,Y 425.285,Z 397.51,A -85,B 0,C 180,E1 -9945.283,E2 -9945.283} C_VEL
LIN {X 0,Y 425.276,Z 397.513,A -85,B 0,C 180,E1 -9948.621,E2 -9948.621} C_VEL
LIN {X 0,Y 425.311,Z 397.507,A -85,B 0,C 180,E1 -9951.103,E2 -9951.103} C_VEL
LIN {X 0,Y 425.302,Z 397.51,A -85,B 0,C 180,E1 -9954.664,E2 -9954.664} C_VEL
LIN {X 0,Y 425.267,Z 397.513,A -85,B 0,C 180,E1 -9958.073,E2 -9958.073} C_VEL
LIN {X 0,Y 425.333,Z 397.502,A -85,B 0,C 180,E1 -9961.368,E2 -9961.368} C_VEL
LIN {X 0,Y 425.298,Z 397.511,A -85,B 0,C 180,E1 -9964.555,E2 -9964.555} C_VEL
LIN {X 0,Y 425.29,Z 397.508,A -85,B 0,C 180,E1 -9967.661,E2 -9967.661} C_VEL
LIN {X 0,Y 425.364,Z 397.501,A -85,B 0,C 180,E1 -9970.704,E2 -9970.704} C_VEL
LIN {X 0,Y 425.391,Z 397.495,A -85,B 0,C 180,E1 -9973.688,E2 -9973.688} C_VEL
LIN {X 0,Y 425.414,Z 397.493,A -85,B 0,C 180,E1 -9977.598,E2 -9977.598} C_VEL
LIN {X 0,Y 425.444,Z 397.489,A -85,B 0,C 180,E1 -9981.45,E2 -9981.45} C_VEL
LIN {X 0,Y 425.556,Z 397.478,A -85,B 0,C 180,E1 -9984.313,E2 -9984.313} C_VEL
LIN {X 0,Y 425.575,Z 397.475,A -85,B 0,C 180,E1 -9988.107,E2 -9988.107} C_VEL
LIN {X 0,Y 425.704,Z 397.46,A -85,B 0,C 180,E1 -9990,E2 -9990} C_VEL
LIN {X 0,Y 425.558,Z 397.477,A -85,B 0,C 180,E1 -9992.839,E2 -9992.839} C_VEL
LIN {X 0,Y 425.531,Z 397.48,A -85,B 0,C 180,E1 -9995.687,E2 -9995.687} C_VEL
LIN {X 0,Y 425.187,Z 397.525,A -85,B 0,C 180,E1 -9998.555,E2 -9998.555} C_VEL
LIN {X 0,Y 425.1,Z 397.698,A -85,B 0,C 180,E1 -9999.135,E2 -9999.135} C_VEL
LIN {X 0,Y 424.738,Z 398.083,A -85,B 0,C 180,E1 -9999.662,E2 -9999.662} C_VEL
LIN {X 0,Y 422.751,Z 399.478,A -85,B 0,C 180,E1 -10000.683,E2 -10000.683} C_VEL
LIN {X 0,Y 418.997,Z 401.753,A -85,B 0,C 180,E1 -10002.197,E2 -10002.197} C_VEL
LIN {X 0,Y 417.914,Z 402.794,A -85,B 0,C 180,E1 -10002.984,E2 -10002.984} C_VEL
LIN {X 0,Y 417.81,Z 403.124,A -85,B 0,C 180,E1 -10003.252,E2 -10003.252} C_VEL
LIN {X 0,Y 417.648,Z 407.258,A -85,B 0,C 180,E1 -10006.622,E2 -10006.622} C_VEL
LIN {X 0,Y 417.455,Z 411.073,A -85,B 0,C 180,E1 -10009.676,E2 -10009.676} C_VEL
LIN {X 0,Y 417.334,Z 415.048,A -85,B 0,C 180,E1 -10012.788,E2 -10012.788} C_VEL
LIN {X 0,Y 417.272,Z 419.074,A -85,B 0,C 180,E1 -10015.903,E2 -10015.903} C_VEL
LIN {X 0,Y 420.728,Z 434.63,A -85,B 0,C 180,E1 -10016.599,E2 -10016.599} C_VEL
LIN {X 0,Y 421.996,Z 441.624,A -85,B 0,C 180,E1 -10016.99,E2 -10016.99} C_VEL
LIN {X 0,Y 421.316,Z 454.336,A -85,B 0,C 180,E1 -10017.757,E2 -10017.757} C_VEL
LIN {X 0,Y 420.686,Z 464.734,A -85,B 0,C 180,E1 -10018.568,E2 -10018.568} C_VEL
LIN {X 0,Y 420.105,Z 474.888,A -85,B 0,C 180,E1 -10019.551,E2 -10019.551} C_VEL
LIN {X 0,Y 419.406,Z 484.785,A -85,B 0,C 180,E1 -10020.736,E2 -10020.736} C_VEL
LIN {X 0,Y 418.849,Z 492.808,A -85,B 0,C 180,E1 -10021.907,E2 -10021.907} C_VEL
LIN {X 0,Y 418.285,Z 500.365,A -85,B 0,C 180,E1 -10023.245,E2 -10023.245} C_VEL
LIN {X 0,Y 417.903,Z 506.218,A -85,B 0,C 180,E1 -10024.508,E2 -10024.508} C_VEL
LIN {X 0,Y 417.522,Z 512.15,A -85,B 0,C 180,E1 -10026.102,E2 -10026.102} C_VEL
LIN {X 0,Y 417.269,Z 516.596,A -85,B 0,C 180,E1 -10027.663,E2 -10027.663} C_VEL
LIN {X 0,Y 417.067,Z 519.751,A -85,B 0,C 180,E1 -10029.182,E2 -10029.182} C_VEL
LIN {X 0,Y 416.911,Z 522.209,A -85,B 0,C 180,E1 -10031.104,E2 -10031.104} C_VEL
LIN {X 0,Y 416.897,Z 522.996,A -85,B 0,C 180,E1 -10032.4,E2 -10032.4} C_VEL
LIN {X 0,Y 416.914,Z 523.034,A -85,B 0,C 180,E1 -10033.72,E2 -10033.72} C_VEL
LIN {X 0,Y 416.944,Z 522.305,A -85,B 0,C 180,E1 -10035.068,E2 -10035.068} C_VEL
LIN {X 0,Y 417.056,Z 520.781,A -85,B 0,C 180,E1 -10036.436,E2 -10036.436} C_VEL
LIN {X 0,Y 417.224,Z 518.378,A -85,B 0,C 180,E1 -10037.83,E2 -10037.83} C_VEL
LIN {X 0,Y 417.427,Z 514.968,A -85,B 0,C 180,E1 -10039.256,E2 -10039.256} C_VEL
LIN {X 0,Y 417.743,Z 510.416,A -85,B 0,C 180,E1 -10040.704,E2 -10040.704} C_VEL
LIN {X 0,Y 418.155,Z 504.515,A -85,B 0,C 180,E1 -10042.178,E2 -10042.178} C_VEL
LIN {X 0,Y 418.685,Z 496.992,A -85,B 0,C 180,E1 -10043.679,E2 -10043.679} C_VEL
LIN {X 0,Y 419.329,Z 489.027,A -85,B 0,C 180,E1 -10044.964,E2 -10044.964} C_VEL
LIN {X 0,Y 420.061,Z 479.652,A -85,B 0,C 180,E1 -10046.199,E2 -10046.199} C_VEL
LIN {X 0,Y 420.805,Z 469.612,A -85,B 0,C 180,E1 -10047.268,E2 -10047.268} C_VEL
LIN {X 0,Y 421.488,Z 458.126,A -85,B 0,C 180,E1 -10048.252,E2 -10048.252} C_VEL
LIN {X 0,Y 422.086,Z 448.172,A -85,B 0,C 180,E1 -10048.924,E2 -10048.924} C_VEL
LIN {X 0,Y 422.225,Z 440.881,A -85,B 0,C 180,E1 -10049.339,E2 -10049.339} C_VEL
LIN {X 0,Y 419.571,Z 428.503,A -85,B 0,C 180,E1 -10050.007,E2 -10050.007} C_VEL
LIN {X 0,Y 417.385,Z 419.916,A -85,B 0,C 180,E1 -10050.39,E2 -10050.39} C_VEL
LIN {X 0,Y 417.499,Z 415.425,A -85,B 0,C 180,E1 -10054.045,E2 -10054.045} C_VEL
LIN {X 0,Y 417.63,Z 412.842,A -85,B 0,C 180,E1 -10056.179,E2 -10056.179} C_VEL
LIN {X 0,Y 417.795,Z 409.126,A -85,B 0,C 180,E1 -10059.313,E2 -10059.313} C_VEL
LIN {X 0,Y 417.983,Z 405.566,A -85,B 0,C 180,E1 -10062.383,E2 -10062.383} C_VEL
LIN {X 0,Y 418.146,Z 402.177,A -85,B 0,C 180,E1 -10065.397,E2 -10065.397} C_VEL
LIN {X 0,Y 418.311,Z 399.972,A -85,B 0,C 180,E1 -10067.384,E2 -10067.384} C_VEL
LIN {X 0,Y 418.254,Z 398.93,A -85,B 0,C 180,E1 -10068.367,E2 -10068.367} C_VEL
LIN {X 0,Y 418.267,Z 398.389,A -85,B 0,C 180,E1 -10069.349,E2 -10069.349} C_VEL
LIN {X 0,Y 418.509,Z 398.358,A -85,B 0,C 180,E1 -10072.279,E2 -10072.279} C_VEL
LIN {X 0,Y 418.509,Z 398.356,A -85,B 0,C 180,E1 -10074.217,E2 -10074.217} C_VEL
LIN {X 0,Y 418.541,Z 398.353,A -85,B 0,C 180,E1 -10078.076,E2 -10078.076} C_VEL
LIN {X 0,Y 418.67,Z 398.336,A -85,B 0,C 180,E1 -10080,E2 -10080} C_VEL
LIN {X 0,Y 418.506,Z 398.357,A -85,B 0,C 180,E1 -10082.888,E2 -10082.888} C_VEL
LIN {X 0,Y 418.49,Z 398.359,A -85,B 0,C 180,E1 -10086.751,E2 -10086.751} C_VEL
LIN {X 0,Y 418.337,Z 398.377,A -85,B 0,C 180,E1 -10089.672,E2 -10089.672} C_VEL
LIN {X 0,Y 418.342,Z 398.377,A -85,B 0,C 180,E1 -10093.001,E2 -10093.001} C_VEL
LIN {X 0,Y 418.309,Z 398.381,A -85,B 0,C 180,E1 -10096.736,E2 -10096.736} C_VEL
LIN {X 0,Y 418.267,Z 398.385,A -85,B 0,C 180,E1 -10099.791,E2 -10099.791} C_VEL
LIN {X 0,Y 418.234,Z 398.391,A -85,B 0,C 180,E1 -10102.736,E2 -10102.736} C_VEL
LIN {X 0,Y 418.268,Z 398.386,A -85,B 0,C 180,E1 -10105.904,E2 -10105.904} C_VEL
LIN {X 0,Y 418.271,Z 398.385,A -85,B 0,C 180,E1 -10109.162,E2 -10109.162} C_VEL
LIN {X 0,Y 418.255,Z 398.388,A -85,B 0,C 180,E1 -10112.845,E2 -10112.845} C_VEL
LIN {X 0,Y 418.246,Z 398.391,A -85,B 0,C 180,E1 -10116.239,E2 -10116.239} C_VEL
LIN {X 0,Y 418.264,Z 398.388,A -85,B 0,C 180,E1 -10119.681,E2 -10119.681} C_VEL
LIN {X 0,Y 418.243,Z 398.391,A -85,B 0,C 180,E1 -10122.324,E2 -10122.324} C_VEL
LIN {X 0,Y 418.234,Z 398.391,A -85,B 0,C 180,E1 -10125.109,E2 -10125.109} C_VEL
LIN {X 0,Y 418.255,Z 398.395,A -85,B 0,C 180,E1 -10127.77,E2 -10127.77} C_VEL
LIN {X 0,Y 419.006,Z 402.543,A -85,B 0,C 180,E1 -10130.494,E2 -10130.494} C_VEL
LIN {X 0,Y 419.703,Z 407.554,A -85,B 0,C 180,E1 -10133.492,E2 -10133.492} C_VEL
LIN {X 0,Y 419.657,Z 411.904,A -85,B 0,C 180,E1 -10135.874,E2 -10135.874} C_VEL
LIN {X 0,Y 419.118,Z 417.575,A -85,B 0,C 180,E1 -10138.782,E2 -10138.782} C_VEL
LIN {X 0,Y 418.583,Z 424.051,A -85,B 0,C 180,E1 -10141.959,E2 -10141.959} C_VEL
LIN {X 0,Y 418.21,Z 430.802,A -85,B 0,C 180,E1 -10145.158,E2 -10145.158} C_VEL
LIN {X 0,Y 417.892,Z 437.656,A -85,B 0,C 180,E1 -10148.286,E2 -10148.286} C_VEL
LIN {X 0,Y 417.527,Z 445.715,A -85,B 0,C 180,E1 -10151.857,E2 -10151.857} C_VEL
LIN {X 0,Y 417.512,Z 447.596,A -85,B 0,C 180,E1 -10152.622,E2 -10152.622} C_VEL
LIN {X 0,Y 419.932,Z 461.154,A -85,B 0,C 180,E1 -10153.154,E2 -10153.154} C_VEL
LIN {X 0,Y 421.485,Z 474.231,A -85,B 0,C 180,E1 -10153.845,E2 -10153.845} C_VEL
LIN {X 0,Y 421.532,Z 479.452,A -85,B 0,C 180,E1 -10154.157,E2 -10154.157} C_VEL
LIN {X 0,Y 420.732,Z 491.514,A -85,B 0,C 180,E1 -10154.995,E2 -10154.995} C_VEL
LIN {X 0,Y 419.948,Z 502.643,A -85,B 0,C 180,E1 -10155.985,E2 -10155.985} C_VEL
LIN {X 0,Y 419.324,Z 513.24,A -85,B 0,C 180,E1 -10157.17,E2 -10157.17} C_VEL
LIN {X 0,Y 418.613,Z 522.093,A -85,B 0,C 180,E1 -10158.378,E2 -10158.378} C_VEL
LIN {X 0,Y 417.997,Z 530.739,A -85,B 0,C 180,E1 -10159.832,E2 -10159.832} C_VEL
LIN {X 0,Y 417.572,Z 537.674,A -85,B 0,C 180,E1 -10161.288,E2 -10161.288} C_VEL
LIN {X 0,Y 417.275,Z 543.24,A -85,B 0,C 180,E1 -10162.743,E2 -10162.743} C_VEL
LIN {X 0,Y 417.112,Z 547.61,A -85,B 0,C 180,E1 -10164.198,E2 -10164.198} C_VEL
LIN {X 0,Y 417.111,Z 549.932,A -85,B 0,C 180,E1 -10165.168,E2 -10165.168} C_VEL
LIN {X 0,Y 417.019,Z 551.801,A -85,B 0,C 180,E1 -10166.135,E2 -10166.135} C_VEL
LIN {X 0,Y 417.033,Z 553.208,A -85,B 0,C 180,E1 -10167.102,E2 -10167.102} C_VEL
LIN {X 0,Y 417.07,Z 554.217,A -85,B 0,C 180,E1 -10168.069,E2 -10168.069} C_VEL
LIN {X 0,Y 417.032,Z 554.832,A -85,B 0,C 180,E1 -10169.035,E2 -10169.035} C_VEL
LIN {X 0,Y 417.026,Z 555.035,A -85,B 0,C 180,E1 -10170,E2 -10170} C_VEL
LIN {X 0,Y 417.071,Z 554.191,A -85,B 0,C 180,E1 -10171.932,E2 -10171.932} C_VEL
LIN {X 0,Y 417.047,Z 553.178,A -85,B 0,C 180,E1 -10172.898,E2 -10172.898} C_VEL
LIN {X 0,Y 417.019,Z 551.739,A -85,B 0,C 180,E1 -10173.866,E2 -10173.866} C_VEL
LIN {X 0,Y 417.127,Z 548.754,A -85,B 0,C 180,E1 -10175.317,E2 -10175.317} C_VEL
LIN {X 0,Y 417.233,Z 544.704,A -85,B 0,C 180,E1 -10176.772,E2 -10176.772} C_VEL
LIN {X 0,Y 417.507,Z 538.466,A -85,B 0,C 180,E1 -10178.47,E2 -10178.47} C_VEL
LIN {X 0,Y 417.913,Z 531.671,A -85,B 0,C 180,E1 -10179.926,E2 -10179.926} C_VEL
LIN {X 0,Y 418.455,Z 523.225,A -85,B 0,C 180,E1 -10181.382,E2 -10181.382} C_VEL
LIN {X 0,Y 419.097,Z 514.528,A -85,B 0,C 180,E1 -10182.592,E2 -10182.592} C_VEL
LIN {X 0,Y 419.722,Z 503.976,A -85,B 0,C 180,E1 -10183.789,E2 -10183.789} C_VEL
LIN {X 0,Y 420.458,Z 493.231,A -85,B 0,C 180,E1 -10184.768,E2 -10184.768} C_VEL
LIN {X 0,Y 421.2,Z 481.49,A -85,B 0,C 180,E1 -10185.605,E2 -10185.605} C_VEL
LIN {X 0,Y 421.432,Z 475.46,A -85,B 0,C 180,E1 -10185.96,E2 -10185.96} C_VEL
LIN {X 0,Y 419.809,Z 462.342,A -85,B 0,C 180,E1 -10186.645,E2 -10186.645} C_VEL
LIN {X 0,Y 417.626,Z 449.211,A -85,B 0,C 180,E1 -10187.145,E2 -10187.145} C_VEL
LIN {X 0,Y 417.521,Z 448.256,A -85,B 0,C 180,E1 -10187.171,E2 -10187.171} C_VEL
LIN {X 0,Y 417.814,Z 440.27,A -85,B 0,C 180,E1 -10190.686,E2 -10190.686} C_VEL
LIN {X 0,Y 418.084,Z 433.36,A -85,B 0,C 180,E1 -10193.794,E2 -10193.794} C_VEL
LIN {X 0,Y 418.478,Z 426.118,A -85,B 0,C 180,E1 -10197.115,E2 -10197.115} C_VEL
LIN {X 0,Y 418.931,Z 419.549,A -85,B 0,C 180,E1 -10200.217,E2 -10200.217} C_VEL
LIN {X 0,Y 419.373,Z 413.637,A -85,B 0,C 180,E1 -10203.079,E2 -10203.079} C_VEL
LIN {X 0,Y 419.677,Z 409.181,A -85,B 0,C 180,E1 -10205.316,E2 -10205.316} C_VEL
LIN {X 0,Y 419.494,Z 405.774,A -85,B 0,C 180,E1 -10207.094,E2 -10207.094} C_VEL
LIN {X 0,Y 418.598,Z 400.057,A -85,B 0,C 180,E1 -10210.255,E2 -10210.255} C_VEL
LIN {X 0,Y 418.273,Z 398.385,A -85,B 0,C 180,E1 -10211.261,E2 -10211.261} C_VEL
LIN {X 0,Y 418.237,Z 398.39,A -85,B 0,C 180,E1 -10215.109,E2 -10215.109} C_VEL
LIN {X 0,Y 418.241,Z 398.388,A -85,B 0,C 180,E1 -10217.767,E2 -10217.767} C_VEL
LIN {X 0,Y 418.25,Z 398.386,A -85,B 0,C 180,E1 -10220.62,E2 -10220.62} C_VEL
LIN {X 0,Y 418.245,Z 398.386,A -85,B 0,C 180,E1 -10223.976,E2 -10223.976} C_VEL
LIN {X 0,Y 418.258,Z 398.387,A -85,B 0,C 180,E1 -10227.156,E2 -10227.156} C_VEL
LIN {X 0,Y 418.269,Z 398.385,A -85,B 0,C 180,E1 -10230.895,E2 -10230.895} C_VEL
LIN {X 0,Y 418.271,Z 398.382,A -85,B 0,C 180,E1 -10234.096,E2 -10234.096} C_VEL
LIN {X 0,Y 418.239,Z 398.39,A -85,B 0,C 180,E1 -10237.264,E2 -10237.264} C_VEL
LIN {X 0,Y 418.284,Z 398.381,A -85,B 0,C 180,E1 -10240.364,E2 -10240.364} C_VEL
LIN {X 0,Y 418.318,Z 398.379,A -85,B 0,C 180,E1 -10243.405,E2 -10243.405} C_VEL
LIN {X 0,Y 418.347,Z 398.377,A -85,B 0,C 180,E1 -10246.999,E2 -10246.999} C_VEL
LIN {X 0,Y 418.342,Z 398.374,A -85,B 0,C 180,E1 -10250.329,E2 -10250.329} C_VEL
LIN {X 0,Y 418.514,Z 398.353,A -85,B 0,C 180,E1 -10252.279,E2 -10252.279} C_VEL
LIN {X 0,Y 418.513,Z 398.353,A -85,B 0,C 180,E1 -10254.217,E2 -10254.217} C_VEL
LIN {X 0,Y 418.542,Z 398.349,A -85,B 0,C 180,E1 -10258.075,E2 -10258.075} C_VEL
LIN {X 0,Y 418.671,Z 398.333,A -85,B 0,C 180,E1 -10260,E2 -10260} C_VEL
LIN {X 0,Y 418.501,Z 398.357,A -85,B 0,C 180,E1 -10262.888,E2 -10262.888} C_VEL
LIN {X 0,Y 418.494,Z 398.357,A -85,B 0,C 180,E1 -10266.751,E2 -10266.751} C_VEL
LIN {X 0,Y 418.401,Z 398.37,A -85,B 0,C 180,E1 -10268.695,E2 -10268.695} C_VEL
LIN {X 0,Y 418.316,Z 398.377,A -85,B 0,C 180,E1 -10271.631,E2 -10271.631} C_VEL
LIN {X 0,Y 418.303,Z 398.382,A -85,B 0,C 180,E1 -10274.597,E2 -10274.597} C_VEL
LIN {X 0,Y 418.289,Z 398.381,A -85,B 0,C 180,E1 -10277.604,E2 -10277.604} C_VEL
LIN {X 0,Y 418.25,Z 398.389,A -85,B 0,C 180,E1 -10280.663,E2 -10280.663} C_VEL
LIN {X 0,Y 418.288,Z 398.38,A -85,B 0,C 180,E1 -10283.781,E2 -10283.781} C_VEL
LIN {X 0,Y 418.311,Z 398.381,A -85,B 0,C 180,E1 -10287.07,E2 -10287.07} C_VEL
LIN {X 0,Y 418.245,Z 398.388,A -85,B 0,C 180,E1 -10290.272,E2 -10290.272} C_VEL
LIN {X 0,Y 418.249,Z 398.385,A -85,B 0,C 180,E1 -10293.677,E2 -10293.677} C_VEL
LIN {X 0,Y 418.241,Z 398.387,A -85,B 0,C 180,E1 -10297.224,E2 -10297.224} C_VEL
LIN {X 0,Y 418.247,Z 398.385,A -85,B 0,C 180,E1 -10299.682,E2 -10299.682} C_VEL
LIN {X 0,Y 418.23,Z 398.39,A -85,B 0,C 180,E1 -10302.321,E2 -10302.321} C_VEL
LIN {X 0,Y 418.236,Z 398.389,A -85,B 0,C 180,E1 -10305.109,E2 -10305.109} C_VEL
LIN {X 0,Y 418.241,Z 398.387,A -85,B 0,C 180,E1 -10307.767,E2 -10307.767} C_VEL
LIN {X 0,Y 418.257,Z 398.387,A -85,B 0,C 180,E1 -10310.619,E2 -10310.619} C_VEL
LIN {X 0,Y 418.247,Z 398.387,A -85,B 0,C 180,E1 -10313.976,E2 -10313.976} C_VEL
LIN {X 0,Y 418.259,Z 398.385,A -85,B 0,C 180,E1 -10317.156,E2 -10317.156} C_VEL
LIN {X 0,Y 418.27,Z 398.384,A -85,B 0,C 180,E1 -10320.895,E2 -10320.895} C_VEL
LIN {X 0,Y 418.273,Z 398.384,A -85,B 0,C 180,E1 -10324.096,E2 -10324.096} C_VEL
LIN {X 0,Y 418.24,Z 398.386,A -85,B 0,C 180,E1 -10327.264,E2 -10327.264} C_VEL
LIN {X 0,Y 418.286,Z 398.384,A -85,B 0,C 180,E1 -10330.364,E2 -10330.364} C_VEL
LIN {X 0,Y 418.319,Z 398.375,A -85,B 0,C 180,E1 -10333.404,E2 -10333.404} C_VEL
LIN {X 0,Y 418.348,Z 398.374,A -85,B 0,C 180,E1 -10336.999,E2 -10336.999} C_VEL
LIN {X 0,Y 418.342,Z 398.377,A -85,B 0,C 180,E1 -10340.328,E2 -10340.328} C_VEL
LIN {X 0,Y 418.515,Z 398.356,A -85,B 0,C 180,E1 -10342.279,E2 -10342.279} C_VEL
LIN {X 0,Y 418.516,Z 398.355,A -85,B 0,C 180,E1 -10344.217,E2 -10344.217} C_VEL
LIN {X 0,Y 418.544,Z 398.351,A -85,B 0,C 180,E1 -10348.075,E2 -10348.075} C_VEL
LIN {X 0,Y 418.673,Z 398.335,A -85,B 0,C 180,E1 -10350,E2 -10350} C_VEL
LIN {X 0,Y 418.512,Z 398.354,A -85,B 0,C 180,E1 -10352.887,E2 -10352.887} C_VEL
LIN {X 0,Y 418.485,Z 398.358,A -85,B 0,C 180,E1 -10355.783,E2 -10355.783} C_VEL
LIN {X 0,Y 418.125,Z 398.404,A -85,B 0,C 180,E1 -10358.7,E2 -10358.7} C_VEL
LIN {X 0,Y 417.991,Z 398.854,A -85,B 0,C 180,E1 -10359.679,E2 -10359.679} C_VEL
LIN {X 0,Y 417.81,Z 403.124,A -85,B 0,C 180,E1 -10363.252,E2 -10363.252} C_VEL
LIN {X 0,Y 417.091,Z 404.157,A -85,B 0,C 180,E1 -10364.043,E2 -10364.043} C_VEL
LIN {X 0,Y 414.168,Z 406.031,A -85,B 0,C 180,E1 -10365.324,E2 -10365.324} C_VEL
LIN {X 0,Y 411.694,Z 407.554,A -85,B 0,C 180,E1 -10366.358,E2 -10366.358} C_VEL
LIN {X 0,Y 410.6,Z 408.651,A -85,B 0,C 180,E1 -10367.159,E2 -10367.159} C_VEL
LIN {X 0,Y 410.492,Z 408.997,A -85,B 0,C 180,E1 -10367.431,E2 -10367.431} C_VEL
LIN {X 0,Y 410.357,Z 412.212,A -85,B 0,C 180,E1 -10370.031,E2 -10370.031} C_VEL
LIN {X 0,Y 410.256,Z 416.198,A -85,B 0,C 180,E1 -10373.203,E2 -10373.203} C_VEL
LIN {X 0,Y 410.181,Z 419.362,A -85,B 0,C 180,E1 -10375.634,E2 -10375.634} C_VEL
LIN {X 0,Y 413.235,Z 432.479,A -85,B 0,C 180,E1 -10376.209,E2 -10376.209} C_VEL
LIN {X 0,Y 415.115,Z 442.882,A -85,B 0,C 180,E1 -10376.792,E2 -10376.792} C_VEL
LIN {X 0,Y 414.473,Z 454.306,A -85,B 0,C 180,E1 -10377.498,E2 -10377.498} C_VEL
LIN {X 0,Y 413.768,Z 465.631,A -85,B 0,C 180,E1 -10378.397,E2 -10378.397} C_VEL
LIN {X 0,Y 413.138,Z 475.852,A -85,B 0,C 180,E1 -10379.419,E2 -10379.419} C_VEL
LIN {X 0,Y 412.475,Z 484.602,A -85,B 0,C 180,E1 -10380.484,E2 -10380.484} C_VEL
LIN {X 0,Y 411.79,Z 494.318,A -85,B 0,C 180,E1 -10381.942,E2 -10381.942} C_VEL
LIN {X 0,Y 411.205,Z 502.37,A -85,B 0,C 180,E1 -10383.448,E2 -10383.448} C_VEL
LIN {X 0,Y 410.662,Z 509.489,A -85,B 0,C 180,E1 -10385.151,E2 -10385.151} C_VEL
LIN {X 0,Y 410.297,Z 514.915,A -85,B 0,C 180,E1 -10386.834,E2 -10386.834} C_VEL
LIN {X 0,Y 410.06,Z 519.267,A -85,B 0,C 180,E1 -10388.723,E2 -10388.723} C_VEL
LIN {X 0,Y 409.837,Z 522.1,A -85,B 0,C 180,E1 -10390.664,E2 -10390.664} C_VEL
LIN {X 0,Y 409.825,Z 523.283,A -85,B 0,C 180,E1 -10392.49,E2 -10392.49} C_VEL
LIN {X 0,Y 409.817,Z 523.273,A -85,B 0,C 180,E1 -10393.924,E2 -10393.924} C_VEL
LIN {X 0,Y 409.859,Z 522.415,A -85,B 0,C 180,E1 -10395.328,E2 -10395.328} C_VEL
LIN {X 0,Y 409.993,Z 520.764,A -85,B 0,C 180,E1 -10396.712,E2 -10396.712} C_VEL
LIN {X 0,Y 410.185,Z 518.348,A -85,B 0,C 180,E1 -10398.07,E2 -10398.07} C_VEL
LIN {X 0,Y 410.475,Z 513.678,A -85,B 0,C 180,E1 -10399.926,E2 -10399.926} C_VEL
LIN {X 0,Y 410.922,Z 507.768,A -85,B 0,C 180,E1 -10401.637,E2 -10401.637} C_VEL
LIN {X 0,Y 411.505,Z 500.373,A -85,B 0,C 180,E1 -10403.291,E2 -10403.291} C_VEL
LIN {X 0,Y 412.17,Z 491.999,A -85,B 0,C 180,E1 -10404.777,E2 -10404.777} C_VEL
LIN {X 0,Y 412.87,Z 483.49,A -85,B 0,C 180,E1 -10405.996,E2 -10405.996} C_VEL
LIN {X 0,Y 413.694,Z 473.234,A -85,B 0,C 180,E1 -10407.192,E2 -10407.192} C_VEL
LIN {X 0,Y 414.439,Z 462.535,A -85,B 0,C 180,E1 -10408.2,E2 -10408.2} C_VEL
LIN {X 0,Y 415.098,Z 451.06,A -85,B 0,C 180,E1 -10409.051,E2 -10409.051} C_VEL
LIN {X 0,Y 415.569,Z 443.239,A -85,B 0,C 180,E1 -10409.512,E2 -10409.512} C_VEL
LIN {X 0,Y 413.185,Z 431.328,A -85,B 0,C 180,E1 -10410.203,E2 -10410.203} C_VEL
LIN {X 0,Y 410.321,Z 420.215,A -85,B 0,C 180,E1 -10410.725,E2 -10410.725} C_VEL
LIN {X 0,Y 410.412,Z 416.777,A -85,B 0,C 180,E1 -10413.562,E2 -10413.562} C_VEL
LIN {X 0,Y 410.619,Z 412.896,A -85,B 0,C 180,E1 -10416.818,E2 -10416.818} C_VEL
LIN {X 0,Y 410.814,Z 408.968,A -85,B 0,C 180,E1 -10420.203,E2 -10420.203} C_VEL
LIN {X 0,Y 411.009,Z 405.529,A -85,B 0,C 180,E1 -10423.246,E2 -10423.246} C_VEL
LIN {X 0,Y 411.28,Z 401.23,A -85,B 0,C 180,E1 -10427.165,E2 -10427.165} C_VEL
LIN {X 0,Y 411.198,Z 399.269,A -85,B 0,C 180,E1 -10429.164,E2 -10429.164} C_VEL
LIN {X 0,Y 411.477,Z 399.234,A -85,B 0,C 180,E1 -10432.147,E2 -10432.147} C_VEL
LIN {X 0,Y 411.471,Z 399.233,A -85,B 0,C 180,E1 -10434.118,E2 -10434.118} C_VEL
LIN {X 0,Y 411.51,Z 399.229,A -85,B 0,C 180,E1 -10438.043,E2 -10438.043} C_VEL
LIN {X 0,Y 411.64,Z 399.212,A -85,B 0,C 180,E1 -10440,E2 -10440} C_VEL
LIN {X 0,Y 411.462,Z 399.234,A -85,B 0,C 180,E1 -10442.937,E2 -10442.937} C_VEL
LIN {X 0,Y 411.456,Z 399.235,A -85,B 0,C 180,E1 -10446.867,E2 -10446.867} C_VEL
LIN {X 0,Y 411.289,Z 399.255,A -85,B 0,C 180,E1 -10449.839,E2 -10449.839} C_VEL
LIN {X 0,Y 411.301,Z 399.254,A -85,B 0,C 180,E1 -10453.104,E2 -10453.104} C_VEL
LIN {X 0,Y 411.259,Z 399.259,A -85,B 0,C 180,E1 -10456.869,E2 -10456.869} C_VEL
LIN {X 0,Y 411.226,Z 399.262,A -85,B 0,C 180,E1 -10459.987,E2 -10459.987} C_VEL
LIN {X 0,Y 411.199,Z 399.266,A -85,B 0,C 180,E1 -10463.148,E2 -10463.148} C_VEL
LIN {X 0,Y 411.235,Z 399.262,A -85,B 0,C 180,E1 -10466.381,E2 -10466.381} C_VEL
LIN {X 0,Y 411.208,Z 399.266,A -85,B 0,C 180,E1 -10469.712,E2 -10469.712} C_VEL
LIN {X 0,Y 411.203,Z 399.267,A -85,B 0,C 180,E1 -10473.156,E2 -10473.156} C_VEL
LIN {X 0,Y 411.193,Z 399.269,A -85,B 0,C 180,E1 -10476.554,E2 -10476.554} C_VEL
LIN {X 0,Y 411.226,Z 399.265,A -85,B 0,C 180,E1 -10479.731,E2 -10479.731} C_VEL
LIN {X 0,Y 411.175,Z 399.271,A -85,B 0,C 180,E1 -10483.134,E2 -10483.134} C_VEL
LIN {X 0,Y 411.166,Z 399.27,A -85,B 0,C 180,E1 -10485.882,E2 -10485.882} C_VEL
LIN {X 0,Y 411.175,Z 399.283,A -85,B 0,C 180,E1 -10487.385,E2 -10487.385} C_VEL
LIN {X 0,Y 411.936,Z 403.35,A -85,B 0,C 180,E1 -10490.152,E2 -10490.152} C_VEL
LIN {X 0,Y 412.701,Z 408.679,A -85,B 0,C 180,E1 -10493.415,E2 -10493.415} C_VEL
LIN {X 0,Y 412.653,Z 412.96,A -85,B 0,C 180,E1 -10495.804,E2 -10495.804} C_VEL
LIN {X 0,Y 411.954,Z 420.583,A -85,B 0,C 180,E1 -10499.784,E2 -10499.784} C_VEL
LIN {X 0,Y 411.34,Z 428.399,A -85,B 0,C 180,E1 -10503.627,E2 -10503.627} C_VEL
LIN {X 0,Y 410.935,Z 436.496,A -85,B 0,C 180,E1 -10507.449,E2 -10507.449} C_VEL
